(* IEC 61131-3 sources: SRCI/RobotLibrary/Library/Functions/Convert/TO_STRING, 78 files *)

(* ---- ABORTING_MODE_TO_STRING.st ---- *)
FUNCTION ABORTING_MODE_TO_STRING : STRING
// -------------------------------------------------------------------------
//  SRCI Robot Library
// -------------------------------------------------------------------------
//
//  Object:      ABORTING_MODE_TO_STRING
//  Author:      Thorsten Brach
//  Date:        2025-02-23
//
//  Description:
//
//
//  Copyright:
//    (C) 2025 Thorsten Brach. All rights reserved
//             Licensed under the LGPL-3.0 license.
//
//  Disclaimer:
//    This project is provided without any guarantee and can be used for
//    private and commercial purposes. Any use is at the user’s
//    own risk and responsibility.
//
// -------------------------------------------------------------------------
VAR_INPUT
  /// AbortingMode
  Value : AbortingMode;
END_VAR

  CASE Value
  OF
    AbortingMode.BUFFER : ABORTING_MODE_TO_STRING := StrReplace('BUFFER ({0})','{0}' , SINT_TO_STRING(Value));
    AbortingMode.ABORT  : ABORTING_MODE_TO_STRING := StrReplace('ABORT ({0})' ,'{0}' , SINT_TO_STRING(Value));
  ELSE
    ABORTING_MODE_TO_STRING := CONCAT('ABORTING_MODE_TO_STRING Function: Error -> no parsing for value ', SINT_TO_STRING(Value));
  END_CASE

END_FUNCTION

(* ---- ALARM_MESSAGE_TO_STRING.st ---- *)
FUNCTION ALARM_MESSAGE_TO_STRING : STRING(RobotLibraryParameter.MESSAGE_TEXT_LEN)
// -------------------------------------------------------------------------
//  SRCI Robot Library
// -------------------------------------------------------------------------
//
//  Object:      ALARM_MESSAGE_TO_STRING
//  Author:      Thorsten Brach
//  Date:        2025-03-31
//
//  Description:
//
//
//  Copyright:
//    (C) 2025 Thorsten Brach. All rights reserved
//             Licensed under the LGPL-3.0 license.
//
//  Disclaimer:
//    This project is provided without any guarantee and can be used for
//    private and commercial purposes. Any use is at the user’s
//    own risk and responsibility.
//
// -------------------------------------------------------------------------
VAR_INPUT
  /// AlarmMessag
  Message : AlarmMessage;
END_VAR
VAR CONSTANT
  /// Carrage return and line feed
  CRLF       : STRING := '$R$N';
END_VAR

  ALARM_MESSAGE_TO_STRING := CONCAT    (ALARM_MESSAGE_TO_STRING, DATE_TO_STRING(Message.Timestamp.SystemDate));
  ALARM_MESSAGE_TO_STRING := CONCAT    (ALARM_MESSAGE_TO_STRING, '-');
  ALARM_MESSAGE_TO_STRING := CONCAT    (ALARM_MESSAGE_TO_STRING, TOD_TO_STRING (Message.Timestamp.SystemTime));
  ALARM_MESSAGE_TO_STRING := StrReplace(ALARM_MESSAGE_TO_STRING, 'TOD#','' );
  ALARM_MESSAGE_TO_STRING := StrReplace(ALARM_MESSAGE_TO_STRING, 'D#', '' );
  ALARM_MESSAGE_TO_STRING := CONCAT    (ALARM_MESSAGE_TO_STRING, ':');
  ALARM_MESSAGE_TO_STRING := CONCAT    (ALARM_MESSAGE_TO_STRING, MESSAGE_TYPE_TO_STRING(Value := Message.MessageType, AlignString := TRUE));
  ALARM_MESSAGE_TO_STRING := CONCAT    (ALARM_MESSAGE_TO_STRING, ':');
  ALARM_MESSAGE_TO_STRING := CONCAT    (ALARM_MESSAGE_TO_STRING, SEVERITY_TO_STRING    ( Value := Message.Severity  , AlignString := TRUE));
  ALARM_MESSAGE_TO_STRING := CONCAT    (ALARM_MESSAGE_TO_STRING, ':');
  ALARM_MESSAGE_TO_STRING := CONCAT    (ALARM_MESSAGE_TO_STRING, DWORD_TO_STRING(Message.MessageCode));
  ALARM_MESSAGE_TO_STRING := CONCAT    (ALARM_MESSAGE_TO_STRING, ':');
  ALARM_MESSAGE_TO_STRING := CONCAT    (ALARM_MESSAGE_TO_STRING, Message.MessageText);
  ALARM_MESSAGE_TO_STRING := CONCAT    (ALARM_MESSAGE_TO_STRING, CRLF);

END_FUNCTION

(* ---- AREA_TYPE_TO_STRING.st ---- *)
FUNCTION AREA_TYPE_TO_STRING : STRING
// -------------------------------------------------------------------------
//  SRCI Robot Library
// -------------------------------------------------------------------------
//
//  Object:      AREA_TYPE_TO_STRING
//  Author:      Thorsten Brach
//  Date:        2025-02-01
//
//  Description:
//
//
//  Copyright:
//    (C) 2025 Thorsten Brach. All rights reserved
//             Licensed under the LGPL-3.0 license.
//
//  Disclaimer:
//    This project is provided without any guarantee and can be used for
//    private and commercial purposes. Any use is at the user’s
//    own risk and responsibility.
//
// -------------------------------------------------------------------------
VAR_INPUT
  /// AreaType
  Value : AreaType;
END_VAR

  CASE Value
  OF
    AreaType.AXES     : AREA_TYPE_TO_STRING := StrReplace('AXES ({0})'     ,'{0}' , USINT_TO_STRING(Value));
    AreaType.BOX      : AREA_TYPE_TO_STRING := StrReplace('BOX ({0})'      ,'{0}' , USINT_TO_STRING(Value));
    AreaType.CYLINDER : AREA_TYPE_TO_STRING := StrReplace('CYLINDER ({0})' ,'{0}' , USINT_TO_STRING(Value));
    AreaType.SPHERE   : AREA_TYPE_TO_STRING := StrReplace('SPHERE ({0})'   ,'{0}' , USINT_TO_STRING(Value));
  ELSE
    AREA_TYPE_TO_STRING := CONCAT('AREA_TYPE_TO_STRING Function: Error -> no parsing for value ', USINT_TO_STRING(Value));
  END_CASE

END_FUNCTION

(* ---- ARM_CONFIG_ELBOW_TO_STRING.st ---- *)
FUNCTION ARM_CONFIG_ELBOW_TO_STRING : STRING
// -------------------------------------------------------------------------
//  SRCI Robot Library
// -------------------------------------------------------------------------
//
//  Object:      ARM_CONFIG_ELBOW_TO_STRING
//  Author:      Thorsten Brach
//  Date:        2025-02-04
//
//  Description:
//
//
//  Copyright:
//    (C) 2025 Thorsten Brach. All rights reserved
//             Licensed under the LGPL-3.0 license.
//
//  Disclaimer:
//    This project is provided without any guarantee and can be used for
//    private and commercial purposes. Any use is at the user’s
//    own risk and responsibility.
//
// -------------------------------------------------------------------------
VAR_INPUT
  /// ArmConfigElbow
  Value : ArmConfigElbow;
END_VAR

  CASE Value
  OF
    ArmConfigElbow.USE_CONFIG : ARM_CONFIG_ELBOW_TO_STRING := StrReplace('Elbow = USE_CONFIG ({0})','{0}' , INT_TO_STRING(Value));
    ArmConfigElbow.SAME       : ARM_CONFIG_ELBOW_TO_STRING := StrReplace('Elbow = SAME ({0})'      ,'{0}' , INT_TO_STRING(Value));
    ArmConfigElbow.FREE       : ARM_CONFIG_ELBOW_TO_STRING := StrReplace('Elbow = FREE ({0})'      ,'{0}' , INT_TO_STRING(Value));
    ArmConfigElbow.DOWN       : ARM_CONFIG_ELBOW_TO_STRING := StrReplace('Elbow = DOWN ({0})'      ,'{0}' , INT_TO_STRING(Value));
    ArmConfigElbow.UP         : ARM_CONFIG_ELBOW_TO_STRING := StrReplace('Elbow = UP ({0})'        ,'{0}' , INT_TO_STRING(Value));
  ELSE
    ARM_CONFIG_ELBOW_TO_STRING := CONCAT('ARM_CONFIG_ELBOW_TO_STRING Function: Error -> no parsing for value ', INT_TO_STRING(Value));
  END_CASE

END_FUNCTION

(* ---- ARM_CONFIG_SHOULDER_TO_STRING.st ---- *)
FUNCTION ARM_CONFIG_SHOULDER_TO_STRING : STRING
// -------------------------------------------------------------------------
//  SRCI Robot Library
// -------------------------------------------------------------------------
//
//  Object:      ARM_CONFIG_SHOULDER_TO_STRING
//  Author:      Thorsten Brach
//  Date:        2025-02-04
//
//  Description:
//
//
//  Copyright:
//    (C) 2025 Thorsten Brach. All rights reserved
//             Licensed under the LGPL-3.0 license.
//
//  Disclaimer:
//    This project is provided without any guarantee and can be used for
//    private and commercial purposes. Any use is at the user’s
//    own risk and responsibility.
//
// -------------------------------------------------------------------------
VAR_INPUT
  /// ArmConfigShoulder
  Value : ArmConfigShoulder;
END_VAR

  CASE Value
  OF
    ArmConfigShoulder.USE_CONFIG : ARM_CONFIG_SHOULDER_TO_STRING := StrReplace('Shoulder = USE_CONFIG ({0})','{0}' , INT_TO_STRING(Value));
    ArmConfigShoulder.SAME       : ARM_CONFIG_SHOULDER_TO_STRING := StrReplace('Shoulder = SAME ({0})'      ,'{0}' , INT_TO_STRING(Value));
    ArmConfigShoulder.FREE       : ARM_CONFIG_SHOULDER_TO_STRING := StrReplace('Shoulder = FREE ({0})'      ,'{0}' , INT_TO_STRING(Value));
    ArmConfigShoulder.BACK       : ARM_CONFIG_SHOULDER_TO_STRING := StrReplace('Shoulder = BACK ({0})'      ,'{0}' , INT_TO_STRING(Value));
    ArmConfigShoulder.FRONT      : ARM_CONFIG_SHOULDER_TO_STRING := StrReplace('Shoulder = FRONT ({0})'     ,'{0}' , INT_TO_STRING(Value));
  ELSE
    ARM_CONFIG_SHOULDER_TO_STRING := CONCAT('ARM_CONFIG_SHOULDER_TO_STRING Function: Error -> no parsing for value ', INT_TO_STRING(Value));
  END_CASE

END_FUNCTION

(* ---- ARM_CONFIG_TO_STRING.st ---- *)
FUNCTION ARM_CONFIG_TO_STRING : STRING
// -------------------------------------------------------------------------
//  SRCI Robot Library
// -------------------------------------------------------------------------
//
//  Object:      ARM_CONFIG_TO_STRING
//  Author:      Thorsten Brach
//  Date:        2025-01-23
//
//  Description:
//
//
//  Copyright:
//    (C) 2025 Thorsten Brach. All rights reserved
//             Licensed under the LGPL-3.0 license.
//
//  Disclaimer:
//    This project is provided without any guarantee and can be used for
//    private and commercial purposes. Any use is at the user’s
//    own risk and responsibility.
//
// -------------------------------------------------------------------------
VAR_INPUT
  /// ArmConfigParameter
  Value : ArmConfigParameter;
END_VAR

VAR
  /// temporary byte
 _tmpByte : BYTE;
END_VAR

  Value := Value;

  _tmpByte.0 := Value.Shoulder = ArmConfigShoulder.USE_CONFIG;
  _tmpByte.1 := Value.Elbow    = ArmConfigElbow   .USE_CONFIG;
  _tmpByte.2 := Value.Wrist    = ArmConfigWrist   .USE_CONFIG;

  ARM_CONFIG_TO_STRING := BYTE_TO_STRING_BIN(_tmpByte);

END_FUNCTION

(* ---- ARM_CONFIG_WRIST_TO_STRING.st ---- *)
FUNCTION ARM_CONFIG_WRIST_TO_STRING : STRING
// -------------------------------------------------------------------------
//  SRCI Robot Library
// -------------------------------------------------------------------------
//
//  Object:      ARM_CONFIG_WRIST_TO_STRING
//  Author:      Thorsten Brach
//  Date:        2025-02-04
//
//  Description:
//
//
//  Copyright:
//    (C) 2025 Thorsten Brach. All rights reserved
//             Licensed under the LGPL-3.0 license.
//
//  Disclaimer:
//    This project is provided without any guarantee and can be used for
//    private and commercial purposes. Any use is at the user’s
//    own risk and responsibility.
//
// -------------------------------------------------------------------------
VAR_INPUT
  /// ArmConfigWrist
  Value : ArmConfigWrist;
END_VAR

  CASE Value
  OF
    ArmConfigWrist.USE_CONFIG : ARM_CONFIG_WRIST_TO_STRING := StrReplace('Wrist = USE_CONFIG ({0})','{0}' , INT_TO_STRING(Value));
    ArmConfigWrist.SAME       : ARM_CONFIG_WRIST_TO_STRING := StrReplace('Wrist = SAME ({0})'      ,'{0}' , INT_TO_STRING(Value));
    ArmConfigWrist.FREE       : ARM_CONFIG_WRIST_TO_STRING := StrReplace('Wrist = FREE ({0})'      ,'{0}' , INT_TO_STRING(Value));
    ArmConfigWrist.FLIP       : ARM_CONFIG_WRIST_TO_STRING := StrReplace('Wrist = FLIP ({0})'      ,'{0}' , INT_TO_STRING(Value));
    ArmConfigWrist.NON_FLIP   : ARM_CONFIG_WRIST_TO_STRING := StrReplace('Wrist = NON_FLIP ({0})'  ,'{0}' , INT_TO_STRING(Value));
  ELSE
    ARM_CONFIG_WRIST_TO_STRING := CONCAT('ARM_CONFIG_WRIST_TO_STRING Function: Error -> no parsing for value ', INT_TO_STRING(Value));
  END_CASE

END_FUNCTION

(* ---- BLENDING_MODE_TO_STRING.st ---- *)
FUNCTION BLENDING_MODE_TO_STRING : STRING
// -------------------------------------------------------------------------
//  SRCI Robot Library
// -------------------------------------------------------------------------
//
//  Object:      BLENDING_MODE_TO_STRING
//  Author:      Thorsten Brach
//  Date:        2025-01-23
//
//  Description:
//
//
//  Copyright:
//    (C) 2025 Thorsten Brach. All rights reserved
//             Licensed under the LGPL-3.0 license.
//
//  Disclaimer:
//    This project is provided without any guarantee and can be used for
//    private and commercial purposes. Any use is at the user’s
//    own risk and responsibility.
//
// -------------------------------------------------------------------------
VAR_INPUT
  /// BlendingMode
  Value : BlendingMode;
END_VAR

  CASE Value
  OF
    BlendingMode.EXACT_STOP           : BLENDING_MODE_TO_STRING := StrReplace('EXACT_STOP ({0})','{0}'           , USINT_TO_STRING(Value));
    BlendingMode.DEFINED_VELOCITY     : BLENDING_MODE_TO_STRING := StrReplace('DEFINED_VELOCITY ({0})','{0}'     , USINT_TO_STRING(Value));
    BlendingMode.CORNER_DISTANCE      : BLENDING_MODE_TO_STRING := StrReplace('CORNER_DISTANCE ({0})','{0}'      , USINT_TO_STRING(Value));
    BlendingMode.MAX_CORNER_DEVIATION : BLENDING_MODE_TO_STRING := StrReplace('MAX_CORNER_DEVIATION ({0})','{0}' , USINT_TO_STRING(Value));
    BlendingMode.CORNER_DISTANCE_2R   : BLENDING_MODE_TO_STRING := StrReplace('CORNER_DISTANCE_2R ({0})','{0}'   , USINT_TO_STRING(Value));
    BlendingMode.RAMP_OVERLAP         : BLENDING_MODE_TO_STRING := StrReplace('RAMP_OVERLAP ({0})','{0}'         , USINT_TO_STRING(Value));
    BlendingMode.CORNER_DISTANCE_1R   : BLENDING_MODE_TO_STRING := StrReplace('CORNER_DISTANCE_1R ({0})','{0}'   , USINT_TO_STRING(Value));
  ELSE
    BLENDING_MODE_TO_STRING := CONCAT('BLENDING_MODE_TO_STRING Function: Error -> no parsing for value ', USINT_TO_STRING(Value));
  END_CASE

END_FUNCTION

(* ---- BYTE_TO_STRING_BIN.st ---- *)
FUNCTION BYTE_TO_STRING_BIN : STRING
// -------------------------------------------------------------------------
//  SRCI Robot Library
// -------------------------------------------------------------------------
//
//  Object:      BYTE_TO_STRING_BIN
//  Author:      Thorsten Brach
//  Date:        2025-01-20
//
//  Description:
//    Converts a BYTE to a STRING with binary notation
//
//  Copyright:
//    (C) 2024 Thorsten Brach. All rights reserved
//             Licensed under the LGPL-3.0 license.
//
//  Disclaimer:
//    This project is provided without any guarantee and can be used for
//    private and commercial purposes. Any use is at the user’s
//    own risk and responsibility.
//
// -------------------------------------------------------------------------
VAR_INPUT
 /// Value to convert
 Value : BYTE;
END_VAR

  BYTE_TO_STRING_BIN := '2#';

  IF (Value.7)
  THEN
    BYTE_TO_STRING_BIN := CONCAT(BYTE_TO_STRING_BIN, '1');
  ELSE
    BYTE_TO_STRING_BIN := CONCAT(BYTE_TO_STRING_BIN, '0');
  END_IF

  IF (Value.6)
  THEN
    BYTE_TO_STRING_BIN := CONCAT(BYTE_TO_STRING_BIN, '1');
  ELSE
    BYTE_TO_STRING_BIN := CONCAT(BYTE_TO_STRING_BIN, '0');
  END_IF

  IF (Value.5)
  THEN
    BYTE_TO_STRING_BIN := CONCAT(BYTE_TO_STRING_BIN, '1');
  ELSE
    BYTE_TO_STRING_BIN := CONCAT(BYTE_TO_STRING_BIN, '0');
  END_IF

  IF (Value.4)
  THEN
    BYTE_TO_STRING_BIN := CONCAT(BYTE_TO_STRING_BIN, '1_');
  ELSE
    BYTE_TO_STRING_BIN := CONCAT(BYTE_TO_STRING_BIN, '0_');
  END_IF

  IF (Value.3)
  THEN
    BYTE_TO_STRING_BIN := CONCAT(BYTE_TO_STRING_BIN, '1');
  ELSE
    BYTE_TO_STRING_BIN := CONCAT(BYTE_TO_STRING_BIN, '0');
  END_IF

  IF (Value.2)
  THEN
    BYTE_TO_STRING_BIN := CONCAT(BYTE_TO_STRING_BIN, '1');
  ELSE
    BYTE_TO_STRING_BIN := CONCAT(BYTE_TO_STRING_BIN, '0');
  END_IF

  IF (Value.1)
  THEN
    BYTE_TO_STRING_BIN := CONCAT(BYTE_TO_STRING_BIN, '1');
  ELSE
    BYTE_TO_STRING_BIN := CONCAT(BYTE_TO_STRING_BIN, '0');
  END_IF

  IF (Value.0)
  THEN
    BYTE_TO_STRING_BIN := CONCAT(BYTE_TO_STRING_BIN, '1');
  ELSE
    BYTE_TO_STRING_BIN := CONCAT(BYTE_TO_STRING_BIN, '0');
  END_IF

  BYTE_TO_STRING_BIN := CONCAT(BYTE_TO_STRING_BIN, ' (');
  BYTE_TO_STRING_BIN := CONCAT(BYTE_TO_STRING_BIN, WORD_TO_STRING(Value));
  BYTE_TO_STRING_BIN := CONCAT(BYTE_TO_STRING_BIN, ')');

END_FUNCTION

(* ---- CIRC_MODE_TO_STRING.st ---- *)
FUNCTION CIRC_MODE_TO_STRING : STRING
// -------------------------------------------------------------------------
//  SRCI Robot Library
// -------------------------------------------------------------------------
//
//  Object:      CIRC_MODE_TO_STRING
//  Author:      Thorsten Brach
//  Date:        2025-01-30
//
//  Description:
//
//
//  Copyright:
//    (C) 2025 Thorsten Brach. All rights reserved
//             Licensed under the LGPL-3.0 license.
//
//  Disclaimer:
//    This project is provided without any guarantee and can be used for
//    private and commercial purposes. Any use is at the user’s
//    own risk and responsibility.
//
// -------------------------------------------------------------------------
VAR_INPUT
  /// CircMode
  Value : CircMode;
END_VAR

  CASE Value
  OF
    CircMode.BORDER            : CIRC_MODE_TO_STRING := StrReplace('BORDER ({0})'            ,'{0}' , SINT_TO_STRING(Value));
    CircMode.CENTER            : CIRC_MODE_TO_STRING := StrReplace('CENTER ({0})'            ,'{0}' , SINT_TO_STRING(Value));
    CircMode.CENTER_WITH_ANGLE : CIRC_MODE_TO_STRING := StrReplace('CENTER_WITH_ANGLE ({0})' ,'{0}' , SINT_TO_STRING(Value));
    CircMode.RADIUS            : CIRC_MODE_TO_STRING := StrReplace('RADIUS ({0})'            ,'{0}' , SINT_TO_STRING(Value));
  ELSE
    CIRC_MODE_TO_STRING := CONCAT('CIRC_MODE_TO_STRING Function: Error -> no parsing for value ', SINT_TO_STRING(Value));
  END_CASE

END_FUNCTION

(* ---- CIRC_PLANE_TO_STRING.st ---- *)
FUNCTION CIRC_PLANE_TO_STRING : STRING
// -------------------------------------------------------------------------
//  SRCI Robot Library
// -------------------------------------------------------------------------
//
//  Object:      CIRC_PLANE_TO_STRING
//  Author:      Thorsten Brach
//  Date:        2025-01-30
//
//  Description:
//
//
//  Copyright:
//    (C) 2025 Thorsten Brach. All rights reserved
//             Licensed under the LGPL-3.0 license.
//
//  Disclaimer:
//    This project is provided without any guarantee and can be used for
//    private and commercial purposes. Any use is at the user’s
//    own risk and responsibility.
//
// -------------------------------------------------------------------------
VAR_INPUT
  /// CircPlane
  Value : CircPlane;
END_VAR

  CASE Value
  OF
    CircPlane.XZ_PLANE : CIRC_PLANE_TO_STRING := StrReplace('XZ_PLANE ({0})' ,'{0}' , SINT_TO_STRING(Value));
    CircPlane.YZ_PLANE : CIRC_PLANE_TO_STRING := StrReplace('YZ_PLANE ({0})' ,'{0}' , SINT_TO_STRING(Value));
    CircPlane.XY_PLANE : CIRC_PLANE_TO_STRING := StrReplace('XY_PLANE ({0})' ,'{0}' , SINT_TO_STRING(Value));
  ELSE
    CIRC_PLANE_TO_STRING := CONCAT('CIRC_PLANE_TO_STRING Function: Error -> no parsing for value ', SINT_TO_STRING(Value));
  END_CASE

END_FUNCTION

(* ---- CMD_MESSAGE_STATE_TO_STRING.st ---- *)
FUNCTION CMD_MESSAGE_STATE_TO_STRING : STRING
// -------------------------------------------------------------------------
//  SRCI Robot Library
// -------------------------------------------------------------------------
//
//  Object:      CMD_MESSAGE_STATE_TO_STRING
//  Author:      Thorsten Brach
//  Date:        2024-11-16
//
//  Description:
//
//
//  Copyright:
//    (C) 2024 Thorsten Brach. All rights reserved
//             Licensed under the LGPL-3.0 license.
//
//  Disclaimer:
//    This project is provided without any guarantee and can be used for
//    private and commercial purposes. Any use is at the user’s
//    own risk and responsibility.
//
// -------------------------------------------------------------------------
VAR_INPUT
  /// Command message state
  Value : CmdMessageState;
END_VAR

  CASE Value
  OF
    CmdMessageState.EMPTY               : CMD_MESSAGE_STATE_TO_STRING := StrReplace('EMPTY ({0})'              ,'{0}', USINT_TO_STRING(Value));
    CmdMessageState.CREATED             : CMD_MESSAGE_STATE_TO_STRING := StrReplace('CREATED ({0})'            ,'{0}', USINT_TO_STRING(Value));
    CmdMessageState.BUFFERED            : CMD_MESSAGE_STATE_TO_STRING := StrReplace('BUFFERED ({0})'           ,'{0}', USINT_TO_STRING(Value));
    CmdMessageState.BUFFERED_IN_PLANNER : CMD_MESSAGE_STATE_TO_STRING := StrReplace('BUFFERED_IN_PLANNER ({0})','{0}', USINT_TO_STRING(Value));
    CmdMessageState.ACTIVE              : CMD_MESSAGE_STATE_TO_STRING := StrReplace('ACTIVE ({0})'             ,'{0}', USINT_TO_STRING(Value));
    CmdMessageState.INTERRUPTED         : CMD_MESSAGE_STATE_TO_STRING := StrReplace('INTERRUPTED ({0})'        ,'{0}', USINT_TO_STRING(Value));
    CmdMessageState.ABORT_REQUEST       : CMD_MESSAGE_STATE_TO_STRING := StrReplace('ABORT_REQUEST ({0})'      ,'{0}', USINT_TO_STRING(Value));
    CmdMessageState.DONE                : CMD_MESSAGE_STATE_TO_STRING := StrReplace('DONE ({0})'               ,'{0}', USINT_TO_STRING(Value));
    CmdMessageState.ABORTED             : CMD_MESSAGE_STATE_TO_STRING := StrReplace('ABORTED ({0})'            ,'{0}', USINT_TO_STRING(Value));
    CmdMessageState.ERROR               : CMD_MESSAGE_STATE_TO_STRING := StrReplace('ERROR ({0})'              ,'{0}', USINT_TO_STRING(Value));
  ELSE
    CMD_MESSAGE_STATE_TO_STRING := CONCAT('CMD_MESSAGE_STATE_TO_STRING Function: Error -> no parsing for value ', USINT_TO_STRING(Value));
  END_CASE

END_FUNCTION

(* ---- CMD_TYPE_TO_STRING.st ---- *)
FUNCTION CMD_TYPE_TO_STRING : String
// -------------------------------------------------------------------------
//  SRCI Robot Library
// -------------------------------------------------------------------------
//
//  Object:      CMD_TYPE_TO_STRING
//  Author:      Thorsten Brach
//  Date:        2024-11-16
//
//  Description:
//
//
//  Copyright:
//    (C) 2024 Thorsten Brach. All rights reserved
//             Licensed under the LGPL-3.0 license.
//
//  Disclaimer:
//    This project is provided without any guarantee and can be used for
//    private and commercial purposes. Any use is at the user’s
//    own risk and responsibility.
//
// -------------------------------------------------------------------------
VAR_INPUT
  /// command type
  Value : CmdType;
END_VAR

  CASE Value
  OF
    CmdType.RobotTask                   : CMD_TYPE_TO_STRING := StrReplace('RobotTask ({0})','{0}'                  , UINT_TO_STRING(CmdType.RobotTask));

    CmdType.ReadRobotData               : CMD_TYPE_TO_STRING := StrReplace('ReadRobotData ({0})','{0}'              , UINT_TO_STRING(CmdType.ReadRobotData));

    CmdType.EnableRobot                 : CMD_TYPE_TO_STRING := StrReplace('EnableRobot ({0})','{0}'                , UINT_TO_STRING(CmdType.EnableRobot));

    CmdType.GroupReset                  : CMD_TYPE_TO_STRING := StrReplace('GroupReset ({0})','{0}'                 , UINT_TO_STRING(CmdType.GroupReset));

    CmdType.ReadActualPosition          : CMD_TYPE_TO_STRING := StrReplace('ReadActualPosition ({0})','{0}'         , UINT_TO_STRING(CmdType.ReadActualPosition));

    CmdType.ReadActualPositionCyclic    : CMD_TYPE_TO_STRING := StrReplace('ReadActualPositionCyclic ({0})','{0}'   , UINT_TO_STRING(CmdType.ReadActualPositionCyclic));

    CmdType.ReadDHParameter             : CMD_TYPE_TO_STRING := StrReplace('ReadDHParameter ({0})','{0}'            , UINT_TO_STRING(CmdType.ReadDHParameter));

    CmdType.RestartController           : CMD_TYPE_TO_STRING := StrReplace('RestartController ({0})','{0}'          , UINT_TO_STRING(CmdType.RestartController));

    CmdType.ReadActualTCPVelocity       : CMD_TYPE_TO_STRING := StrReplace('ReadActualTCPVelocity ({0})','{0}'      , UINT_TO_STRING(CmdType.ReadActualTCPVelocity));

    CmdType.UserLogin                   : CMD_TYPE_TO_STRING := StrReplace('UserLogin ({0})','{0}'                  , UINT_TO_STRING(CmdType.UserLogin));

    CmdType.SwitchLanguage              : CMD_TYPE_TO_STRING := StrReplace('SwitchLanguage ({0})','{0}'             , UINT_TO_STRING(CmdType.SwitchLanguage));

    CmdType.ExchangeConfiguration       : CMD_TYPE_TO_STRING := StrReplace('ExchangeConfiguration ({0})','{0}'      , UINT_TO_STRING(CmdType.ExchangeConfiguration));

    CmdType.SetSequence                 : CMD_TYPE_TO_STRING := StrReplace('SetSequence ({0})','{0}'                , UINT_TO_STRING(CmdType.SetSequence));

    CmdType.ChangeSpeedOverride         : CMD_TYPE_TO_STRING := StrReplace('ChangeSpeedOverride ({0})','{0}'        , UINT_TO_STRING(CmdType.ChangeSpeedOverride));

    CmdType.ReadMessages                : CMD_TYPE_TO_STRING := StrReplace('ReadMessages ({0})','{0}'               , UINT_TO_STRING(CmdType.ReadMessages));

    CmdType.ReadRobotReferenceDynamics  : CMD_TYPE_TO_STRING := StrReplace('ReadRobotReferenceDynamics ({0})','{0}' , UINT_TO_STRING(CmdType.ReadRobotReferenceDynamics));

    CmdType.WriteFrameData              : CMD_TYPE_TO_STRING := StrReplace('WriteFrameData ({0})','{0}'             , UINT_TO_STRING(CmdType.WriteFrameData));

    CmdType.WriteToolData               : CMD_TYPE_TO_STRING := StrReplace('WriteToolData ({0})','{0}'              , UINT_TO_STRING(CmdType.WriteToolData));

    CmdType.WriteLoadData               : CMD_TYPE_TO_STRING := StrReplace('WriteLoadData ({0})','{0}'              , UINT_TO_STRING(CmdType.WriteLoadData));

    CmdType.WriteRobotReferenceDynamics : CMD_TYPE_TO_STRING := StrReplace('WriteRobotReferenceDynamics ({0})','{0}', UINT_TO_STRING(CmdType.WriteRobotReferenceDynamics));

    CmdType.WriteRobotDefaultDynamics   : CMD_TYPE_TO_STRING := StrReplace('WriteRobotDefaultDynamics ({0})'  ,'{0}', UINT_TO_STRING(CmdType.WriteRobotDefaultDynamics));

    CmdType.ReadRobotDefaultDynamics    : CMD_TYPE_TO_STRING := StrReplace('ReadRobotDefaultDynamics ({0})'   ,'{0}', UINT_TO_STRING(CmdType.ReadRobotDefaultDynamics));

    CmdType.ReadFrameData               : CMD_TYPE_TO_STRING := StrReplace('ReadFrameData ({0})'              ,'{0}', UINT_TO_STRING(CmdType.ReadFrameData));

    CmdType.ReadToolData                : CMD_TYPE_TO_STRING := StrReplace('ReadToolData ({0})','{0}'               , UINT_TO_STRING(CmdType.ReadToolData));

    CmdType.ReadLoadData                : CMD_TYPE_TO_STRING := StrReplace('ReadLoadData ({0})','{0}'               , UINT_TO_STRING(CmdType.ReadLoadData));

    CmdType.ReadRobotSWLimits           : CMD_TYPE_TO_STRING := StrReplace('ReadRobotSWLimits ({0})','{0}'          , UINT_TO_STRING(CmdType.ReadRobotSWLimits));

    CmdType.WriteRobotSWLimits          : CMD_TYPE_TO_STRING := StrReplace('WriteRobotSWLimits ({0})','{0}'         , UINT_TO_STRING(CmdType.WriteRobotSWLimits));

    CmdType.SetOperationMode            : CMD_TYPE_TO_STRING := StrReplace('SetOperationMode ({0})','{0}'           , UINT_TO_STRING(CmdType.SetOperationMode));

    CmdType.ReadWorkArea                : CMD_TYPE_TO_STRING := StrReplace('ReadWorkArea ({0})','{0}'               , UINT_TO_STRING(CmdType.ReadWorkArea));

    CmdType.WriteWorkArea               : CMD_TYPE_TO_STRING := StrReplace('WriteWorkArea ({0})','{0}'              , UINT_TO_STRING(CmdType.WriteWorkArea));

    CmdType.ActivateWorkArea            : CMD_TYPE_TO_STRING := StrReplace('ActivateWorkArea ({0})','{0}'           , UINT_TO_STRING(CmdType.ActivateWorkArea));

    CmdType.MonitorWorkArea             : CMD_TYPE_TO_STRING := StrReplace('MonitorWorkArea ({0})','{0}'            , UINT_TO_STRING(CmdType.MonitorWorkArea));

    CmdType.GroupJog                    : CMD_TYPE_TO_STRING := StrReplace('GroupJog ({0})','{0}'                   , UINT_TO_STRING(CmdType.GroupJog));

    CmdType.MoveLinearAbsolute          : CMD_TYPE_TO_STRING := StrReplace('MoveLinearAbsolute ({0})','{0}'         , UINT_TO_STRING(CmdType.MoveLinearAbsolute));

    CmdType.MoveDirectAbsolute          : CMD_TYPE_TO_STRING := StrReplace('MoveDirectAbsolute ({0})','{0}'         , UINT_TO_STRING(CmdType.MoveDirectAbsolute));

    CmdType.MoveAxesAbsolute            : CMD_TYPE_TO_STRING := StrReplace('MoveAxesAbsolute ({0})','{0}'           , UINT_TO_STRING(CmdType.MoveAxesAbsolute));

    CmdType.GroupStop                   : CMD_TYPE_TO_STRING := StrReplace('GroupStop ({0})','{0}'                  , UINT_TO_STRING(CmdType.GroupStop));

    CmdType.GroupInterrupt              : CMD_TYPE_TO_STRING := StrReplace('GroupInterrupt ({0})','{0}'             , UINT_TO_STRING(CmdType.GroupInterrupt));

    CmdType.GroupContinue               : CMD_TYPE_TO_STRING := StrReplace('GroupContinue ({0})','{0}'              , UINT_TO_STRING(CmdType.GroupContinue));

    CmdType.MoveLinearRelative          : CMD_TYPE_TO_STRING := StrReplace('MoveLinearRelative ({0})','{0}'         , UINT_TO_STRING(CmdType.MoveLinearRelative));

    CmdType.MoveDirectRelative          : CMD_TYPE_TO_STRING := StrReplace('MoveDirectRelative ({0})','{0}'         , UINT_TO_STRING(CmdType.MoveDirectRelative));

    CmdType.MoveAxesRelative            : CMD_TYPE_TO_STRING := StrReplace('MoveAxesRelative ({0})','{0}'           , UINT_TO_STRING(CmdType.MoveAxesRelative));

    CmdType.ReturnToPrimary             : CMD_TYPE_TO_STRING := StrReplace('ReturnToPrimary ({0})','{0}'            , UINT_TO_STRING(CmdType.ReturnToPrimary));

    CmdType.MoveCircularAbsolute        : CMD_TYPE_TO_STRING := StrReplace('MoveCircularAbsolute ({0})','{0}'       , UINT_TO_STRING(CmdType.MoveCircularAbsolute));

    CmdType.MoveCircularRelative        : CMD_TYPE_TO_STRING := StrReplace('MoveCircularRelative ({0})','{0}'       , UINT_TO_STRING(CmdType.MoveCircularRelative));

    CmdType.MoveLinearOffset            : CMD_TYPE_TO_STRING := StrReplace('MoveLinearOffset ({0})','{0}'           , UINT_TO_STRING(CmdType.MoveLinearOffset));

    CmdType.MoveDirectOffset            : CMD_TYPE_TO_STRING := StrReplace('MoveDirectOffset ({0})','{0}'           , UINT_TO_STRING(CmdType.MoveDirectOffset));

    CmdType.WaitTime                    : CMD_TYPE_TO_STRING := StrReplace('WaitTime ({0})','{0}'                   , UINT_TO_STRING(CmdType.WaitTime));

    CmdType.MoveApproachLinear          : CMD_TYPE_TO_STRING := StrReplace('MoveApproachLinear ({0})','{0}'         , UINT_TO_STRING(CmdType.MoveApproachLinear));

    CmdType.MoveDepartLinear            : CMD_TYPE_TO_STRING := StrReplace('MoveDepartLinear ({0})','{0}'           , UINT_TO_STRING(CmdType.MoveDepartLinear));

    CmdType.MoveApproachDirect          : CMD_TYPE_TO_STRING := StrReplace('MoveApproachDirect ({0})','{0}'         , UINT_TO_STRING(CmdType.MoveApproachDirect));

    CmdType.MoveDepartDirect            : CMD_TYPE_TO_STRING := StrReplace('MoveDepartDirect ({0})','{0}'           , UINT_TO_STRING(CmdType.MoveDepartDirect));

    CmdType.SearchHardstop              : CMD_TYPE_TO_STRING := StrReplace('SearchHardstop ({0})','{0}'             , UINT_TO_STRING(CmdType.SearchHardstop));

    CmdType.SearchHardstopJ             : CMD_TYPE_TO_STRING := StrReplace('SearchHardstopJ ({0})','{0}'            , UINT_TO_STRING(CmdType.SearchHardstopJ));

    CmdType.MovePickPlaceLinear         : CMD_TYPE_TO_STRING := StrReplace('MovePickPlaceLinear ({0})','{0}'        , UINT_TO_STRING(CmdType.MovePickPlaceLinear));

    CmdType.MovePickPlaceDirect         : CMD_TYPE_TO_STRING := StrReplace('MovePickPlaceDirect ({0})','{0}'        , UINT_TO_STRING(CmdType.MovePickPlaceDirect));

    CmdType.ActivateConveyorTracking    : CMD_TYPE_TO_STRING := StrReplace('ActivateConveyorTracking ({0})','{0}'   , UINT_TO_STRING(CmdType.ActivateConveyorTracking));

    CmdType.RedefineTrackingPos         : CMD_TYPE_TO_STRING := StrReplace('RedefineTrackingPos ({0})','{0}'        , UINT_TO_STRING(CmdType.RedefineTrackingPos));

    CmdType.SyncToConveyor              : CMD_TYPE_TO_STRING := StrReplace('SyncToConveyor ({0})','{0}'             , UINT_TO_STRING(CmdType.SyncToConveyor));

    CmdType.ConfigureConveyor           : CMD_TYPE_TO_STRING := StrReplace('ConfigureConveyor ({0})','{0}'          , UINT_TO_STRING(CmdType.ConfigureConveyor));

    CmdType.MoveSuperImposed            : CMD_TYPE_TO_STRING := StrReplace('MoveSuperImposed ({0})','{0}'           , UINT_TO_STRING(CmdType.MoveSuperImposed));

    CmdType.MoveSuperImposedDynamic     : CMD_TYPE_TO_STRING := StrReplace('MoveSuperImposedDynamic ({0})','{0}'    , UINT_TO_STRING(CmdType.MoveSuperImposedDynamic));

    CmdType.ReadDigitalInputs           : CMD_TYPE_TO_STRING := StrReplace('ReadDigitalInputs ({0})','{0}'          , UINT_TO_STRING(CmdType.ReadDigitalInputs));

    CmdType.ReadDigitalOutputs          : CMD_TYPE_TO_STRING := StrReplace('ReadDigitalOutputs ({0})','{0}'         , UINT_TO_STRING(CmdType.ReadDigitalOutputs));

    CmdType.WriteDigitalOutputs         : CMD_TYPE_TO_STRING := StrReplace('WriteDigitalOutputs ({0})','{0}'        , UINT_TO_STRING(CmdType.WriteDigitalOutputs));

    CmdType.ReadIntegers                : CMD_TYPE_TO_STRING := StrReplace('ReadIntegers ({0})','{0}'               , UINT_TO_STRING(CmdType.ReadIntegers));

    CmdType.ReadReals                   : CMD_TYPE_TO_STRING := StrReplace('ReadReals ({0})','{0}'                  , UINT_TO_STRING(CmdType.ReadReals));

    CmdType.WriteIntegers               : CMD_TYPE_TO_STRING := StrReplace('WriteIntegers ({0})','{0}'              , UINT_TO_STRING(CmdType.WriteIntegers));

    CmdType.WriteReals                  : CMD_TYPE_TO_STRING := StrReplace('WriteReals ({0})','{0}'                 , UINT_TO_STRING(CmdType.WriteReals));

    CmdType.MoveLinearCam               : CMD_TYPE_TO_STRING := StrReplace('MoveLinearCam ({0})','{0}'              , UINT_TO_STRING(CmdType.MoveLinearCam));

    CmdType.MoveDirectCam               : CMD_TYPE_TO_STRING := StrReplace('MoveDirectCam ({0})','{0}'              , UINT_TO_STRING(CmdType.MoveDirectCam));

    CmdType.MoveCircularCam             : CMD_TYPE_TO_STRING := StrReplace('MoveCircularCam ({0})','{0}'            , UINT_TO_STRING(CmdType.MoveCircularCam));

    CmdType.ReadAnalogInput             : CMD_TYPE_TO_STRING := StrReplace('ReadAnalogInput ({0})','{0}'            , UINT_TO_STRING(CmdType.ReadAnalogInput));

    CmdType.ReadAnalogOutput            : CMD_TYPE_TO_STRING := StrReplace('ReadAnalogOutput ({0})','{0}'           , UINT_TO_STRING(CmdType.ReadAnalogOutput));

    CmdType.WriteAnalogOutput           : CMD_TYPE_TO_STRING := StrReplace('WriteAnalogOutput ({0})','{0}'          , UINT_TO_STRING(CmdType.WriteAnalogOutput));

    CmdType.MeasuringInput              : CMD_TYPE_TO_STRING := StrReplace('MeasuringInput ({0})','{0}'             , UINT_TO_STRING(CmdType.MeasuringInput));

    CmdType.AbortMeasuringInput         : CMD_TYPE_TO_STRING := StrReplace('AbortMeasuringInput ({0})','{0}'        , UINT_TO_STRING(CmdType.AbortMeasuringInput));

    CmdType.SetTriggerRegister          : CMD_TYPE_TO_STRING := StrReplace('SetTriggerRegister ({0})','{0}'         , UINT_TO_STRING(CmdType.SetTriggerRegister));

    CmdType.SetTriggerLimit             : CMD_TYPE_TO_STRING := StrReplace('SetTriggerLimit ({0})','{0}'            , UINT_TO_STRING(CmdType.SetTriggerLimit));

    CmdType.SetTriggerUser              : CMD_TYPE_TO_STRING := StrReplace('SetTriggerUser ({0})','{0}'             , UINT_TO_STRING(CmdType.SetTriggerUser));

    CmdType.SetTriggerError             : CMD_TYPE_TO_STRING := StrReplace('SetTriggerError ({0})','{0}'            , UINT_TO_STRING(CmdType.SetTriggerError));

    CmdType.ReactAtTrigger              : CMD_TYPE_TO_STRING := StrReplace('ReactAtTrigger ({0})','{0}'             , UINT_TO_STRING(CmdType.ReactAtTrigger));

    CmdType.WaitForTrigger              : CMD_TYPE_TO_STRING := StrReplace('WaitForTrigger ({0})','{0}'             , UINT_TO_STRING(CmdType.WaitForTrigger));

    CmdType.ReadSystemVariable          : CMD_TYPE_TO_STRING := StrReplace('ReadSystemVariable ({0})','{0}'         , UINT_TO_STRING(CmdType.ReadSystemVariable));

    CmdType.WriteSystemVariable         : CMD_TYPE_TO_STRING := StrReplace('WriteSystemVariable ({0})','{0}'        , UINT_TO_STRING(CmdType.WriteSystemVariable));

    CmdType.CalculateForwardKinematic   : CMD_TYPE_TO_STRING := StrReplace('CalculateForwardKinematic ({0})','{0}'  , UINT_TO_STRING(CmdType.CalculateForwardKinematic));

    CmdType.CalculateInverseKinematic   : CMD_TYPE_TO_STRING := StrReplace('CalculateInverseKinematic ({0})','{0}'  , UINT_TO_STRING(CmdType.CalculateInverseKinematic));

    CmdType.CalculateCartesianPosition  : CMD_TYPE_TO_STRING := StrReplace('CalculateCartesianPosition ({0})','{0}' , UINT_TO_STRING(CmdType.CalculateCartesianPosition));

    CmdType.CalculateTool               : CMD_TYPE_TO_STRING := StrReplace('CalculateTool ({0})','{0}'              , UINT_TO_STRING(CmdType.CalculateTool));

    CmdType.CalculateFrame              : CMD_TYPE_TO_STRING := StrReplace('CalculateFrame ({0})','{0}'             , UINT_TO_STRING(CmdType.CalculateFrame));

    CmdType.ActivateNextCommand         : CMD_TYPE_TO_STRING := StrReplace('ActivateNextCommand ({0})','{0}'        , UINT_TO_STRING(CmdType.ActivateNextCommand));

    CmdType.ShiftPosition               : CMD_TYPE_TO_STRING := StrReplace('ShiftPosition ({0})','{0}'              , UINT_TO_STRING(CmdType.ShiftPosition));

    CmdType.SetTriggerMotion            : CMD_TYPE_TO_STRING := StrReplace('SetTriggerMotion ({0})','{0}'           , UINT_TO_STRING(CmdType.SetTriggerMotion));

    CmdType.OpenBrake                   : CMD_TYPE_TO_STRING := StrReplace('OpenBrake ({0})','{0}'                  , UINT_TO_STRING(CmdType.OpenBrake));

    CmdType.CallSubprogram              : CMD_TYPE_TO_STRING := StrReplace('CallSubprogram ({0})','{0}'             , UINT_TO_STRING(CmdType.CallSubprogram));

    CmdType.WriteCallSubprogramCyclic   : CMD_TYPE_TO_STRING := StrReplace('WriteCallSubprogramCyclic ({0})','{0}'  , UINT_TO_STRING(CmdType.WriteCallSubprogramCyclic));

    CmdType.ReadCallSubprogramCyclic    : CMD_TYPE_TO_STRING := StrReplace('ReadCallSubprogramCyclic ({0})','{0}'   , UINT_TO_STRING(CmdType.ReadCallSubprogramCyclic));

    CmdType.StopSubprogram              : CMD_TYPE_TO_STRING := StrReplace('StopSubprogram ({0})','{0}'             , UINT_TO_STRING(CmdType.StopSubprogram));

    CmdType.PathAccuracyMode            : CMD_TYPE_TO_STRING := StrReplace('PathAccuracyMode ({0})','{0}'           , UINT_TO_STRING(CmdType.PathAccuracyMode));

    CmdType.AvoidSingularity            : CMD_TYPE_TO_STRING := StrReplace('AvoidSingularity ({0})','{0}'           , UINT_TO_STRING(CmdType.AvoidSingularity));

    CmdType.ForceControl                : CMD_TYPE_TO_STRING := StrReplace('ForceControl ({0})','{0}'               , UINT_TO_STRING(CmdType.ForceControl));

    CmdType.ForceLimit                  : CMD_TYPE_TO_STRING := StrReplace('ForceLimit ({0})','{0}'                 , UINT_TO_STRING(CmdType.ForceLimit));

    CmdType.ReadActualForce             : CMD_TYPE_TO_STRING := StrReplace('ReadActualForce ({0})','{0}'            , UINT_TO_STRING(CmdType.ReadActualForce));

    CmdType.BrakeTest                   : CMD_TYPE_TO_STRING := StrReplace('BrakeTest ({0})','{0}'                  , UINT_TO_STRING(CmdType.BrakeTest));

    CmdType.SoftSwitchTCP               : CMD_TYPE_TO_STRING := StrReplace('SoftSwitchTCP ({0})','{0}'              , UINT_TO_STRING(CmdType.SoftSwitchTCP));

    CmdType.CreateSpline                : CMD_TYPE_TO_STRING := StrReplace('CreateSpline ({0})','{0}'               , UINT_TO_STRING(CmdType.CreateSpline));

    CmdType.DeleteSpline                : CMD_TYPE_TO_STRING := StrReplace('DeleteSpline ({0})','{0}'               , UINT_TO_STRING(CmdType.DeleteSpline));

    CmdType.MoveSpline                  : CMD_TYPE_TO_STRING := StrReplace('MoveSpline ({0})','{0}'                 , UINT_TO_STRING(CmdType.MoveSpline));

    CmdType.DynamicSpline               : CMD_TYPE_TO_STRING := StrReplace('DynamicSpline ({0})','{0}'              , UINT_TO_STRING(CmdType.DynamicSpline));

    CmdType.LoadMeasurementAutomatic    : CMD_TYPE_TO_STRING := StrReplace('LoadMeasurementAutomatic ({0})','{0}'   , UINT_TO_STRING(CmdType.LoadMeasurementAutomatic));

    CmdType.LoadMeasurementSequential   : CMD_TYPE_TO_STRING := StrReplace('LoadMeasurementSequential ({0})','{0}'  , UINT_TO_STRING(CmdType.LoadMeasurementSequential));

    CmdType.CollisionDetection          : CMD_TYPE_TO_STRING := StrReplace('CollisionDetection ({0})','{0}'         , UINT_TO_STRING(CmdType.CollisionDetection));

    CmdType.FreeDrive                   : CMD_TYPE_TO_STRING := StrReplace('FreeDrive ({0})','{0}'                  , UINT_TO_STRING(CmdType.FreeDrive));

    CmdType.UnitMeasurement             : CMD_TYPE_TO_STRING := StrReplace('UnitMeasurement ({0})','{0}'            , UINT_TO_STRING(CmdType.UnitMeasurement));

  ELSE
    CMD_TYPE_TO_STRING := CONCAT('CMD_TYPE_TO_STRING Function: Error -> no parsing for value',UINT_TO_STRING(Value));
  END_CASE

END_FUNCTION

(* ---- COLLISION_REACTION_MODE_TO_STRING.st ---- *)
FUNCTION COLLISION_REACTION_MODE_TO_STRING : STRING
// -------------------------------------------------------------------------
//  SRCI Robot Library
// -------------------------------------------------------------------------
//
//  Object:      COLLISION_REACTION_MODE_TO_STRING
//  Author:      Thorsten Brach
//  Date:        2025-01-24
//
//  Description:
//
//
//  Copyright:
//    (C) 2025 Thorsten Brach. All rights reserved
//             Licensed under the LGPL-3.0 license.
//
//  Disclaimer:
//    This project is provided without any guarantee and can be used for
//    private and commercial purposes. Any use is at the user’s
//    own risk and responsibility.
//
// -------------------------------------------------------------------------
VAR_INPUT
  /// CollisionReactionMode
  Value : CollisionReactionMode;
END_VAR

  CASE Value
  OF
    CollisionReactionMode.REVERSED_MOVEMENT : COLLISION_REACTION_MODE_TO_STRING := StrReplace('REVERSED_MOVEMENT ({0})','{0}' , USINT_TO_STRING(Value));
    CollisionReactionMode.STANDING_STILL    : COLLISION_REACTION_MODE_TO_STRING := StrReplace('STANDING_STILL ({0})'   ,'{0}' , USINT_TO_STRING(Value));
  ELSE
    COLLISION_REACTION_MODE_TO_STRING := CONCAT('COLLISION_REACTION_MODE_TO_STRING Function: Error -> no parsing for value ', USINT_TO_STRING(Value));
  END_CASE

END_FUNCTION

(* ---- CONNECTION_MODE_TO_STRING.st ---- *)
FUNCTION CONNECTION_MODE_TO_STRING : STRING
// -------------------------------------------------------------------------
//  SRCI Robot Library
// -------------------------------------------------------------------------
//
//  Object:      CONNECTION_MODE_TO_STRING
//  Author:      Thorsten Brach
//  Date:        2025-02-01
//
//  Description:
//
//
//  Copyright:
//    (C) 2025 Thorsten Brach. All rights reserved
//             Licensed under the LGPL-3.0 license.
//
//  Disclaimer:
//    This project is provided without any guarantee and can be used for
//    private and commercial purposes. Any use is at the user’s
//    own risk and responsibility.
//
// -------------------------------------------------------------------------
VAR_INPUT
  /// ConnectionMode
  Value : ConnectionMode;
END_VAR

  CASE Value
  OF
    ConnectionMode.RC_CONNECTED  : CONNECTION_MODE_TO_STRING := StrReplace('RC_CONNECTED ({0})'  ,'{0}' , SINT_TO_STRING(Value));
    ConnectionMode.PLC_CONNECTED : CONNECTION_MODE_TO_STRING := StrReplace('PLC_CONNECTED ({0})' ,'{0}' , SINT_TO_STRING(Value));
  ELSE
    CONNECTION_MODE_TO_STRING := CONCAT('CONNECTION_MODE_TO_STRING Function: Error -> no parsing for value ', SINT_TO_STRING(Value));
  END_CASE

END_FUNCTION

(* ---- CONVEYOR_TYPE_TO_STRING.st ---- *)
FUNCTION CONVEYOR_TYPE_TO_STRING : STRING
// -------------------------------------------------------------------------
//  SRCI Robot Library
// -------------------------------------------------------------------------
//
//  Object:      CONVEYOR_TYPE_TO_STRING
//  Author:      Thorsten Brach
//  Date:        2025-02-01
//
//  Description:
//
//
//  Copyright:
//    (C) 2025 Thorsten Brach. All rights reserved
//             Licensed under the LGPL-3.0 license.
//
//  Disclaimer:
//    This project is provided without any guarantee and can be used for
//    private and commercial purposes. Any use is at the user’s
//    own risk and responsibility.
//
// -------------------------------------------------------------------------
VAR_INPUT
  /// ConveyorType
  Value : ConveyorType;
END_VAR

  CASE Value
  OF
    ConveyorType.LINEAR_CONVEYOR_TRACKING   : CONVEYOR_TYPE_TO_STRING := StrReplace('LINEAR_CONVEYOR_TRACKING ({0})'   ,'{0}' , USINT_TO_STRING(Value));
    ConveyorType.CIRCULAR_CONVEYOR_TRACKING : CONVEYOR_TYPE_TO_STRING := StrReplace('CIRCULAR_CONVEYOR_TRACKING ({0})' ,'{0}' , USINT_TO_STRING(Value));
  ELSE
    CONVEYOR_TYPE_TO_STRING := CONCAT('CONVEYOR_TYPE_TO_STRING Function: Error -> no parsing for value ', USINT_TO_STRING(Value));
  END_CASE

END_FUNCTION

(* ---- DATA_ENABLE_SYNC_TO_STRING.st ---- *)
FUNCTION DATA_ENABLE_SYNC_TO_STRING : STRING
// -------------------------------------------------------------------------
//  SRCI Robot Library
// -------------------------------------------------------------------------
//
//  Object:      DATA_ENABLE_SYNC_TO_STRING
//  Author:      Thorsten Brach
//  Date:        2025-01-24
//
//  Description:
//
//
//  Copyright:
//    (C) 2025 Thorsten Brach. All rights reserved
//             Licensed under the LGPL-3.0 license.
//
//  Disclaimer:
//    This project is provided without any guarantee and can be used for
//    private and commercial purposes. Any use is at the user’s
//    own risk and responsibility.
//
// -------------------------------------------------------------------------
VAR_INPUT
  /// DataEnableSync
  Value : DataEnableSync;
END_VAR

VAR
  /// temporary byte
 _tmpByte : BYTE;
END_VAR

  _tmpByte.0 := Value.EnableSyncTool;
  _tmpByte.1 := Value.EnableSyncFrame;
  _tmpByte.2 := Value.EnableSyncLoad;
  _tmpByte.3 := Value.EnableSyncWorkArea;
  _tmpByte.4 := Value.EnableSyncSWLimits;
  _tmpByte.5 := Value.EnableSyncDefaultDynamics;
  _tmpByte.6 := Value.EnableSyncReferenceDynamics;

  DATA_ENABLE_SYNC_TO_STRING := BYTE_TO_STRING_BIN(_tmpByte);

END_FUNCTION

(* ---- DATA_IN_SYNC_TO_STRING.st ---- *)
FUNCTION DATA_IN_SYNC_TO_STRING : STRING
// -------------------------------------------------------------------------
//  SRCI Robot Library
// -------------------------------------------------------------------------
//
//  Object:      DATA_IN_SYNC_TO_STRING
//  Author:      Thorsten Brach
//  Date:        2025-01-24
//
//  Description:
//
//
//  Copyright:
//    (C) 2025 Thorsten Brach. All rights reserved
//             Licensed under the LGPL-3.0 license.
//
//  Disclaimer:
//    This project is provided without any guarantee and can be used for
//    private and commercial purposes. Any use is at the user’s
//    own risk and responsibility.
//
// -------------------------------------------------------------------------
VAR_INPUT
  /// DataInSync
  Value : DataInSync;
END_VAR

VAR
  /// temporary byte
 _tmpByte : BYTE;
END_VAR

  _tmpByte.0 := Value.ToolsInSync;
  _tmpByte.1 := Value.FramesInSync;
  _tmpByte.2 := Value.LoadsInSync;
  _tmpByte.3 := Value.WorkAreasInSync;
  _tmpByte.4 := Value.SoftwareLimitsInSync;
  _tmpByte.5 := Value.DefaultDynamicsInSync;
  _tmpByte.6 := Value.ReferenceDynamicsInSync;
  _tmpByte.7 := FALSE;

  DATA_IN_SYNC_TO_STRING := BYTE_TO_STRING_BIN(_tmpByte);

END_FUNCTION

(* ---- DATA_TYPE_TO_STRING.st ---- *)
FUNCTION DATA_TYPE_TO_STRING : STRING
// -------------------------------------------------------------------------
//  SRCI Robot Library
// -------------------------------------------------------------------------
//
//  Object:      DATA_TYPE_TO_STRING
//  Author:      Thorsten Brach
//  Date:        2025-03-05
//
//  Description:
//
//
//  Copyright:
//    (C) 2025 Thorsten Brach. All rights reserved
//             Licensed under the LGPL-3.0 license.
//
//  Disclaimer:
//    This project is provided without any guarantee and can be used for
//    private and commercial purposes. Any use is at the user’s
//    own risk and responsibility.
//
// -------------------------------------------------------------------------
VAR_INPUT
  /// DataType
  Value : DataType;
END_VAR

  CASE Value
  OF
    DataType.TYPE_BOOL       : DATA_TYPE_TO_STRING := StrReplace('BOOL ({0})'                ,'{0}' , USINT_TO_STRING(Value));
    DataType.TYPE_BYTE       : DATA_TYPE_TO_STRING := StrReplace('BYTE ({0})'                ,'{0}' , USINT_TO_STRING(Value));
    DataType.TYPE_WORD       : DATA_TYPE_TO_STRING := StrReplace('WORD ({0})'                ,'{0}' , USINT_TO_STRING(Value));
    DataType.TYPE_DWORD      : DATA_TYPE_TO_STRING := StrReplace('DWORD ({0})'               ,'{0}' , USINT_TO_STRING(Value));
    DataType.TYPE_SINT       : DATA_TYPE_TO_STRING := StrReplace('SINT ({0})'                ,'{0}' , USINT_TO_STRING(Value));
    DataType.TYPE_USINT      : DATA_TYPE_TO_STRING := StrReplace('USINT ({0})'               ,'{0}' , USINT_TO_STRING(Value));
    DataType.TYPE_INT        : DATA_TYPE_TO_STRING := StrReplace('INT ({0})'                 ,'{0}' , USINT_TO_STRING(Value));
    DataType.TYPE_UINT       : DATA_TYPE_TO_STRING := StrReplace('UINT ({0})'                ,'{0}' , USINT_TO_STRING(Value));
    DataType.TYPE_DINT       : DATA_TYPE_TO_STRING := StrReplace('DINT ({0})'                ,'{0}' , USINT_TO_STRING(Value));
    DataType.TYPE_UDINT      : DATA_TYPE_TO_STRING := StrReplace('UDINT ({0})'               ,'{0}' , USINT_TO_STRING(Value));
    DataType.TYPE_REAL       : DATA_TYPE_TO_STRING := StrReplace('REAL ({0})'                ,'{0}' , USINT_TO_STRING(Value));
    DataType.TYPE_CHAR       : DATA_TYPE_TO_STRING := StrReplace('CHAR ({0})'                ,'{0}' , USINT_TO_STRING(Value));
    DataType.TYPE_CHAR_ARRAY : DATA_TYPE_TO_STRING := StrReplace('ARRAY[0..3] OF CHAR ({0})' ,'{0}' , USINT_TO_STRING(Value));
  ELSE
    DATA_TYPE_TO_STRING := CONCAT('DATA_TYPE_TO_STRING Function: Error -> no parsing for value ', USINT_TO_STRING(Value));
  END_CASE

END_FUNCTION

(* ---- DEFINITION_MODE_TO_STRING.st ---- *)
FUNCTION DEFINITION_MODE_TO_STRING : STRING
// -------------------------------------------------------------------------
//  SRCI Robot Library
// -------------------------------------------------------------------------
//
//  Object:      DEFINITION_MODE_TO_STRING
//  Author:      Thorsten Brach
//  Date:        2025-02-01
//
//  Description:
//
//
//  Copyright:
//    (C) 2025 Thorsten Brach. All rights reserved
//             Licensed under the LGPL-3.0 license.
//
//  Disclaimer:
//    This project is provided without any guarantee and can be used for
//    private and commercial purposes. Any use is at the user’s
//    own risk and responsibility.
//
// -------------------------------------------------------------------------
VAR_INPUT
  /// DefinitionMode
  Value : DefinitionMode;
END_VAR

  CASE Value
  OF
    DefinitionMode.CENTER : DEFINITION_MODE_TO_STRING := StrReplace('CENTER ({0})','{0}' , USINT_TO_STRING(Value));
    DefinitionMode.FACE   : DEFINITION_MODE_TO_STRING := StrReplace('FACE ({0})'  ,'{0}' , USINT_TO_STRING(Value));
  ELSE
    DEFINITION_MODE_TO_STRING := CONCAT('DEFINITION_MODE_TO_STRING Function: Error -> no parsing for value ', USINT_TO_STRING(Value));
  END_CASE

END_FUNCTION

(* ---- DETECTION_MODE_TO_STRING.st ---- *)
FUNCTION DETECTION_MODE_TO_STRING : STRING
// -------------------------------------------------------------------------
//  SRCI Robot Library
// -------------------------------------------------------------------------
//
//  Object:      DETECTION_MODE_TO_STRING
//  Author:      Thorsten Brach
//  Date:        2025-02-01
//
//  Description:
//
//
//  Copyright:
//    (C) 2025 Thorsten Brach. All rights reserved
//             Licensed under the LGPL-3.0 license.
//
//  Disclaimer:
//    This project is provided without any guarantee and can be used for
//    private and commercial purposes. Any use is at the user’s
//    own risk and responsibility.
//
// -------------------------------------------------------------------------
VAR_INPUT
  /// DetectionMode
  Value : DetectionMode;
END_VAR

  CASE Value
  OF
    DetectionMode.TORQUE             : DETECTION_MODE_TO_STRING := StrReplace('TORQUE ({0})'             ,'{0}' , USINT_TO_STRING(Value));
    DetectionMode.FORCE              : DETECTION_MODE_TO_STRING := StrReplace('FORCE ({0})'              ,'{0}' , USINT_TO_STRING(Value));
    DetectionMode.ELECTRICAL_CURRENT : DETECTION_MODE_TO_STRING := StrReplace('ELECTRICAL_CURRENT ({0})' ,'{0}' , USINT_TO_STRING(Value));
    DetectionMode.FOLLOWING_ERROR    : DETECTION_MODE_TO_STRING := StrReplace('FOLLOWING_ERROR ({0})'    ,'{0}' , USINT_TO_STRING(Value));
  ELSE
    DETECTION_MODE_TO_STRING := CONCAT('DETECTION_MODE_TO_STRING Function: Error -> no parsing for value ', USINT_TO_STRING(Value));
  END_CASE

END_FUNCTION

(* ---- ERROR_REACTION_TO_STRING.st ---- *)
FUNCTION ERROR_REACTION_TO_STRING : STRING
// -------------------------------------------------------------------------
//  SRCI Robot Library
// -------------------------------------------------------------------------
//
//  Object:      ERROR_REACTION_TO_STRING
//  Author:      Thorsten Brach
//  Date:        2025-02-01
//
//  Description:
//
//
//  Copyright:
//    (C) 2025 Thorsten Brach. All rights reserved
//             Licensed under the LGPL-3.0 license.
//
//  Disclaimer:
//    This project is provided without any guarantee and can be used for
//    private and commercial purposes. Any use is at the user’s
//    own risk and responsibility.
//
// -------------------------------------------------------------------------
VAR_INPUT
  /// ErrorReaction
  Value : ErrorReaction;
END_VAR

  CASE Value
  OF
    ErrorReaction.ABORT_AND_MOVE : ERROR_REACTION_TO_STRING := StrReplace('ABORT_AND_MOVE ({0})','{0}' , USINT_TO_STRING(Value));
    ErrorReaction.ABORT          : ERROR_REACTION_TO_STRING := StrReplace('ABORT ({0})'         ,'{0}' , USINT_TO_STRING(Value));
    ErrorReaction.NO_REACTION    : ERROR_REACTION_TO_STRING := StrReplace('NO_REACTION ({0})'   ,'{0}' , USINT_TO_STRING(Value));
  ELSE
    ERROR_REACTION_TO_STRING := CONCAT('ERROR_REACTION_TO_STRING Function: Error -> no parsing for value ', USINT_TO_STRING(Value));
  END_CASE

END_FUNCTION

(* ---- ERROR_TRIGGER_MODE_TO_STRING.st ---- *)
FUNCTION ERROR_TRIGGER_MODE_TO_STRING : STRING
// -------------------------------------------------------------------------
//  SRCI Robot Library
// -------------------------------------------------------------------------
//
//  Object:      ERROR_TRIGGER_MODE_TO_STRING
//  Author:      Thorsten Brach
//  Date:        2025-02-01
//
//  Description:
//
//
//  Copyright:
//    (C) 2025 Thorsten Brach. All rights reserved
//             Licensed under the LGPL-3.0 license.
//
//  Disclaimer:
//    This project is provided without any guarantee and can be used for
//    private and commercial purposes. Any use is at the user’s
//    own risk and responsibility.
//
// -------------------------------------------------------------------------
VAR_INPUT
  /// ErrorTriggerMode
  Value : ErrorTriggerMode;
END_VAR

  CASE Value
  OF
    ErrorTriggerMode.ANY_COMMAND                    : ERROR_TRIGGER_MODE_TO_STRING := StrReplace('ANY_COMMAND ({0})'                    ,'{0}' , SINT_TO_STRING(Value));
    ErrorTriggerMode.GENERAL_COMMANDS               : ERROR_TRIGGER_MODE_TO_STRING := StrReplace('GENERAL_COMMANDS ({0})'               ,'{0}' , SINT_TO_STRING(Value));
    ErrorTriggerMode.ADMINISTRATIVE_COMMANDS        : ERROR_TRIGGER_MODE_TO_STRING := StrReplace('ADMINISTRATIVE_COMMANDS ({0})'        ,'{0}' , SINT_TO_STRING(Value));
    ErrorTriggerMode.MOVE_COMMANDS                  : ERROR_TRIGGER_MODE_TO_STRING := StrReplace('MOVE_COMMANDS ({0})'                  ,'{0}' , SINT_TO_STRING(Value));
    ErrorTriggerMode.PERIPHERY_COMMANDS             : ERROR_TRIGGER_MODE_TO_STRING := StrReplace('PERIPHERY_COMMANDS ({0})'             ,'{0}' , SINT_TO_STRING(Value));
    ErrorTriggerMode.EXTENDED_COMMANDS              : ERROR_TRIGGER_MODE_TO_STRING := StrReplace('EXTENDED_COMMANDS ({0})'              ,'{0}' , SINT_TO_STRING(Value));
    ErrorTriggerMode.SPECIFIC_COMMAND_OR_RI_MESSAGE : ERROR_TRIGGER_MODE_TO_STRING := StrReplace('SPECIFIC_COMMAND_OR_RI_MESSAGE ({0})' ,'{0}' , SINT_TO_STRING(Value));
    ErrorTriggerMode.SPECIFIC_RC_OR_RA_MESSAGE_CODE : ERROR_TRIGGER_MODE_TO_STRING := StrReplace('SPECIFIC_RC_OR_RA_MESSAGE_CODE ({0})' ,'{0}' , SINT_TO_STRING(Value));
    ErrorTriggerMode.ANY_RI_MESSAGE_CODE            : ERROR_TRIGGER_MODE_TO_STRING := StrReplace('ANY_RI_MESSAGE_CODE ({0})'            ,'{0}' , SINT_TO_STRING(Value));
    ErrorTriggerMode.ANY_RC_OR_RA_MESSAGE_CODE      : ERROR_TRIGGER_MODE_TO_STRING := StrReplace('ANY_RC_OR_RA_MESSAGE_CODE ({0})'      ,'{0}' , SINT_TO_STRING(Value));
  ELSE
    ERROR_TRIGGER_MODE_TO_STRING := CONCAT('ERROR_TRIGGER_MODE_TO_STRING Function: Error -> no parsing for value ', SINT_TO_STRING(Value));
  END_CASE

END_FUNCTION

(* ---- EXECUTION_MODE_TO_STRING.st ---- *)
FUNCTION EXECUTION_MODE_TO_STRING : STRING
// -------------------------------------------------------------------------
//  SRCI Robot Library
// -------------------------------------------------------------------------
//
//  Object:      EXECUTION_MODE_TO_STRING
//  Author:      Thorsten Brach
//  Date:        2025-01-20
//
//  Description:
//
//
//  Copyright:
//    (C) 2024 Thorsten Brach. All rights reserved
//             Licensed under the LGPL-3.0 license.
//
//  Disclaimer:
//    This project is provided without any guarantee and can be used for
//    private and commercial purposes. Any use is at the user’s
//    own risk and responsibility.
//
// -------------------------------------------------------------------------
VAR_INPUT
  /// ExecMode
  Value : ExecutionMode;
END_VAR

  CASE Value
  OF
    ExecutionMode.SEQUENCE_PRIMARY                 : EXECUTION_MODE_TO_STRING := StrReplace('SEQUENCE_PRIMARY ({0})'                 ,'{0}', USINT_TO_STRING(Value));
    ExecutionMode.SEQUENCE_ABORT_OTHERS_PRIMARY    : EXECUTION_MODE_TO_STRING := StrReplace('SEQUENCE_ABORT_OTHERS_PRIMARY ({0})'    ,'{0}', USINT_TO_STRING(Value));
    ExecutionMode.PARALLEL                         : EXECUTION_MODE_TO_STRING := StrReplace('PARALLEL ({0})'                         ,'{0}', USINT_TO_STRING(Value));
    ExecutionMode.CONTINUOUS                       : EXECUTION_MODE_TO_STRING := StrReplace('CONTINUOUS ({0})'                       ,'{0}', USINT_TO_STRING(Value));
    ExecutionMode.TRIGGER_MULTIPLE                 : EXECUTION_MODE_TO_STRING := StrReplace('TRIGGER_MULTIPLE ({0})'                 ,'{0}', USINT_TO_STRING(Value));
    ExecutionMode.SEQUENCE_SECONDARY               : EXECUTION_MODE_TO_STRING := StrReplace('SEQUENCE_SECONDARY ({0})'               ,'{0}', USINT_TO_STRING(Value));
    ExecutionMode.SEQUENCE_ABORT_OTHERS_SECONDARY  : EXECUTION_MODE_TO_STRING := StrReplace('SEQUENCE_ABORT_OTHERS_SECONDARY ({0})'  ,'{0}', USINT_TO_STRING(Value));
    ExecutionMode.STOP_PARALLEL_CONTINUOUS_TRIGGER : EXECUTION_MODE_TO_STRING := StrReplace('STOP_PARALLEL_CONTINUOUS_TRIGGER ({0})' ,'{0}', USINT_TO_STRING(Value));
  ELSE
    EXECUTION_MODE_TO_STRING := CONCAT('EXECUTION_MODE_TO_STRING Function: Error -> no parsing for value ', USINT_TO_STRING(Value));
  END_CASE

END_FUNCTION

(* ---- EXTERNAL_AXES_FLAGS_TO_STRING.st ---- *)
FUNCTION EXTERNAL_AXES_FLAGS_TO_STRING : STRING
// -------------------------------------------------------------------------
//  SRCI Robot Library
// -------------------------------------------------------------------------
//
//  Object:      EXTERNAL_AXES_FLAGS_TO_STRING
//  Author:      Thorsten Brach
//  Date:        2025-02-26
//
//  Description:
//
//
//  Copyright:
//    (C) 2025 Thorsten Brach. All rights reserved
//             Licensed under the LGPL-3.0 license.
//
//  Disclaimer:
//    This project is provided without any guarantee and can be used for
//    private and commercial purposes. Any use is at the user’s
//    own risk and responsibility.
//
// -------------------------------------------------------------------------
VAR_INPUT
  /// ExternalAxesFlags
  Value : ExternalAxesFlags;
END_VAR

VAR
 _tmpByte : BYTE;
END_VAR

  _tmpByte.0 := Value.Bit00;
  _tmpByte.1 := Value.AxisE1;
  _tmpByte.2 := Value.AxisE2;
  _tmpByte.3 := Value.AxisE3;
  _tmpByte.4 := Value.AxisE4;
  _tmpByte.5 := Value.AxisE5;
  _tmpByte.6 := Value.AxisE6;
  _tmpByte.7 := Value.Bit07;

  EXTERNAL_AXES_FLAGS_TO_STRING := BYTE_TO_STRING_BIN(_tmpByte);

END_FUNCTION

(* ---- FRAGMENT_ACTION_TO_STRING.st ---- *)
FUNCTION FRAGMENT_ACTION_TO_STRING : STRING
// -------------------------------------------------------------------------
//  SRCI Robot Library
// -------------------------------------------------------------------------
//
//  Object:      FRAGMENT_ACTION_TO_STRING
//  Author:      Thorsten Brach
//  Date:        2024-11-16
//
//  Description:
//
//
//  Copyright:
//    (C) 2024 Thorsten Brach. All rights reserved
//             Licensed under the LGPL-3.0 license.
//
//  Disclaimer:
//    This project is provided without any guarantee and can be used for
//    private and commercial purposes. Any use is at the user’s
//    own risk and responsibility.
//
// -------------------------------------------------------------------------
VAR_INPUT
  /// Fragment action
  FragmentAction : BYTE;
END_VAR

  IF ( FragmentAction.0 )
  THEN
   FRAGMENT_ACTION_TO_STRING := CONCAT(FRAGMENT_ACTION_TO_STRING, ' Complete (Bit 0)');
  END_IF

  IF ( FragmentAction.1 )
  THEN
   FRAGMENT_ACTION_TO_STRING := CONCAT(FRAGMENT_ACTION_TO_STRING, ' Reset (Bit 1)');
  END_IF

  IF ( FragmentAction.2 )
  THEN
   FRAGMENT_ACTION_TO_STRING := CONCAT(FRAGMENT_ACTION_TO_STRING, ' Clear (Bit 2)');
  END_IF

END_FUNCTION

(* ---- FRAME_CALCULATION_MODE_TO_STRING.st ---- *)
FUNCTION FRAME_CALCULATION_MODE_TO_STRING : STRING
// -------------------------------------------------------------------------
//  SRCI Robot Library
// -------------------------------------------------------------------------
//
//  Object:      FRAME_CALCULATION_MODE_TO_STRING
//  Author:      Thorsten Brach
//  Date:        2025-02-01
//
//  Description:
//
//
//  Copyright:
//    (C) 2025 Thorsten Brach. All rights reserved
//             Licensed under the LGPL-3.0 license.
//
//  Disclaimer:
//    This project is provided without any guarantee and can be used for
//    private and commercial purposes. Any use is at the user’s
//    own risk and responsibility.
//
// -------------------------------------------------------------------------
VAR_INPUT
  /// FrameCalculationMode
  Value : FrameCalculationMode;
END_VAR

  CASE Value
  OF
    FrameCalculationMode.THREE_POINT_METHOD : FRAME_CALCULATION_MODE_TO_STRING := StrReplace('THREE_POINT_METHOD ({0})','{0}' , SINT_TO_STRING(Value));
    FrameCalculationMode.FOUR_POINT_METHOD  : FRAME_CALCULATION_MODE_TO_STRING := StrReplace('FOUR_POINT_METHOD ({0})' ,'{0}' , SINT_TO_STRING(Value));
    FrameCalculationMode.ONE_POINT_METHOD   : FRAME_CALCULATION_MODE_TO_STRING := StrReplace('ONE_POINT_METHOD ({0})'  ,'{0}' , SINT_TO_STRING(Value));
  ELSE
    FRAME_CALCULATION_MODE_TO_STRING := CONCAT('FRAME_CALCULATION_MODE_TO_STRING Function: Error -> no parsing for value ', SINT_TO_STRING(Value));
  END_CASE

END_FUNCTION

(* ---- IEC_DATE_TO_STRING.st ---- *)
FUNCTION IEC_DATE_TO_STRING : STRING
// -------------------------------------------------------------------------
//  SRCI Robot Library
// -------------------------------------------------------------------------
//
//  Object:      IEC_DATE_TO_STRING
//  Author:      Thorsten Brach
//  Date:        2025-02-01
//
//  Description:
//
//
//  Copyright:
//    (C) 2025 Thorsten Brach. All rights reserved
//             Licensed under the LGPL-3.0 license.
//
//  Disclaimer:
//    This project is provided without any guarantee and can be used for
//    private and commercial purposes. Any use is at the user’s
//    own risk and responsibility.
//
// -------------------------------------------------------------------------
VAR_INPUT
  /// IEC Date
  Value : IEC_DATE;
END_VAR

VAR
  /// temporary date
 _tmpData : DATE;
END_VAR

  IEC_DATE_TO_STRING := DATE_TO_STRING(IEC_DATE_TO_DATE(Value));

END_FUNCTION

(* ---- IEC_TIME_TO_STRING.st ---- *)
FUNCTION IEC_TIME_TO_STRING : STRING
// -------------------------------------------------------------------------
//  SRCI Robot Library
// -------------------------------------------------------------------------
//
//  Object:      ORI_MODE_TO_STRING
//  Author:      Thorsten Brach
//  Date:        2025-01-24
//
//  Description:
//
//
//  Copyright:
//    (C) 2025 Thorsten Brach. All rights reserved
//             Licensed under the LGPL-3.0 license.
//
//  Disclaimer:
//    This project is provided without any guarantee and can be used for
//    private and commercial purposes. Any use is at the user’s
//    own risk and responsibility.
//
// -------------------------------------------------------------------------
VAR_INPUT
  /// IEC_TIME
  Value : IEC_TIME;
END_VAR
VAR
  /// temporary date
 _tmpData : DATE;
END_VAR

  IEC_TIME_TO_STRING := TOD_TO_STRING(IEC_TIME_TO_TIME(Value));

END_FUNCTION

(* ---- INTERPOLATION_MODE_TO_STRING.st ---- *)
FUNCTION INTERPOLATION_MODE_TO_STRING : STRING
// -------------------------------------------------------------------------
//  SRCI Robot Library
// -------------------------------------------------------------------------
//
//  Object:      INTERPOLATION_MODE_TO_STRING
//  Author:      Thorsten Brach
//  Date:        2025-02-01
//
//  Description:
//
//
//  Copyright:
//    (C) 2025 Thorsten Brach. All rights reserved
//             Licensed under the LGPL-3.0 license.
//
//  Disclaimer:
//    This project is provided without any guarantee and can be used for
//    private and commercial purposes. Any use is at the user’s
//    own risk and responsibility.
//
// -------------------------------------------------------------------------
VAR_INPUT
  /// InterpolationMode
  Value : InterpolationMode;
END_VAR

  CASE Value
  OF
    InterpolationMode.LINEAR_INTERPOLATION : INTERPOLATION_MODE_TO_STRING := StrReplace('LINEAR_INTERPOLATION ({0})' ,'{0}' , USINT_TO_STRING(Value));
    InterpolationMode.DIRECT_INTERPOLATION : INTERPOLATION_MODE_TO_STRING := StrReplace('DIRECT_INTERPOLATION ({0})' ,'{0}' , USINT_TO_STRING(Value));
  ELSE
    INTERPOLATION_MODE_TO_STRING := CONCAT('INTERPOLATION_MODE_TO_STRING Function: Error -> no parsing for value ', USINT_TO_STRING(Value));
  END_CASE

END_FUNCTION

(* ---- JOG_CONTROL_TO_STRING.st ---- *)
FUNCTION JOG_CONTROL_TO_STRING : STRING
// -------------------------------------------------------------------------
//  SRCI Robot Library
// -------------------------------------------------------------------------
//
//  Object:      JOG_CONTROL_TO_STRING
//  Author:      Thorsten Brach
//  Date:        2025-03-01
//
//  Description:
//
//
//  Copyright:
//    (C) 2025 Thorsten Brach. All rights reserved
//             Licensed under the LGPL-3.0 license.
//
//  Disclaimer:
//    This project is provided without any guarantee and can be used for
//    private and commercial purposes. Any use is at the user’s
//    own risk and responsibility.
//
// -------------------------------------------------------------------------
VAR_INPUT
  /// JogControl
  Value : JogControl;
END_VAR

  JOG_CONTROL_TO_STRING := '2#';

  IF (Value.E6_Neg)
  THEN
    JOG_CONTROL_TO_STRING := CONCAT(JOG_CONTROL_TO_STRING, '1');
  ELSE
    JOG_CONTROL_TO_STRING := CONCAT(JOG_CONTROL_TO_STRING, '0');
  END_IF

  IF (Value.E6_Pos)
  THEN
    JOG_CONTROL_TO_STRING := CONCAT(JOG_CONTROL_TO_STRING, '1');
  ELSE
    JOG_CONTROL_TO_STRING := CONCAT(JOG_CONTROL_TO_STRING, '0');
  END_IF

  IF (Value.E5_Neg)
  THEN
    JOG_CONTROL_TO_STRING := CONCAT(JOG_CONTROL_TO_STRING, '1');
  ELSE
    JOG_CONTROL_TO_STRING := CONCAT(JOG_CONTROL_TO_STRING, '0');
  END_IF

  IF (Value.E5_Pos)
  THEN
    JOG_CONTROL_TO_STRING := CONCAT(JOG_CONTROL_TO_STRING, '1_');
  ELSE
    JOG_CONTROL_TO_STRING := CONCAT(JOG_CONTROL_TO_STRING, '0_');
  END_IF

  IF (Value.E4_Neg)
  THEN
    JOG_CONTROL_TO_STRING := CONCAT(JOG_CONTROL_TO_STRING, '1');
  ELSE
    JOG_CONTROL_TO_STRING := CONCAT(JOG_CONTROL_TO_STRING, '0');
  END_IF

  IF (Value.E4_Pos)
  THEN
    JOG_CONTROL_TO_STRING := CONCAT(JOG_CONTROL_TO_STRING, '1');
  ELSE
    JOG_CONTROL_TO_STRING := CONCAT(JOG_CONTROL_TO_STRING, '0');
  END_IF

  IF (Value.E3_Neg)
  THEN
    JOG_CONTROL_TO_STRING := CONCAT(JOG_CONTROL_TO_STRING, '1');
  ELSE
    JOG_CONTROL_TO_STRING := CONCAT(JOG_CONTROL_TO_STRING, '0');
  END_IF

  IF (Value.E3_Pos)
  THEN
    JOG_CONTROL_TO_STRING := CONCAT(JOG_CONTROL_TO_STRING, '1');
  ELSE
    JOG_CONTROL_TO_STRING := CONCAT(JOG_CONTROL_TO_STRING, '0');
  END_IF

  JOG_CONTROL_TO_STRING := CONCAT(JOG_CONTROL_TO_STRING, '_');

  IF (Value.E2_Neg)
  THEN
    JOG_CONTROL_TO_STRING := CONCAT(JOG_CONTROL_TO_STRING, '1');
  ELSE
    JOG_CONTROL_TO_STRING := CONCAT(JOG_CONTROL_TO_STRING, '0');
  END_IF

  IF (Value.E2_Pos)
  THEN
    JOG_CONTROL_TO_STRING := CONCAT(JOG_CONTROL_TO_STRING, '1');
  ELSE
    JOG_CONTROL_TO_STRING := CONCAT(JOG_CONTROL_TO_STRING, '0');
  END_IF

  IF (Value.E1_Neg)
  THEN
    JOG_CONTROL_TO_STRING := CONCAT(JOG_CONTROL_TO_STRING, '1');
  ELSE
    JOG_CONTROL_TO_STRING := CONCAT(JOG_CONTROL_TO_STRING, '0');
  END_IF

  IF (Value.E1_Pos)
  THEN
    JOG_CONTROL_TO_STRING := CONCAT(JOG_CONTROL_TO_STRING, '1');
  ELSE
    JOG_CONTROL_TO_STRING := CONCAT(JOG_CONTROL_TO_STRING, '0');
  END_IF

  IF (Value.Rz_J6_Neg)
  THEN
    JOG_CONTROL_TO_STRING := CONCAT(JOG_CONTROL_TO_STRING, '1');
  ELSE
    JOG_CONTROL_TO_STRING := CONCAT(JOG_CONTROL_TO_STRING, '0');
  END_IF

  IF (Value.Rz_J6_Pos)
  THEN
    JOG_CONTROL_TO_STRING := CONCAT(JOG_CONTROL_TO_STRING, '1');
  ELSE
    JOG_CONTROL_TO_STRING := CONCAT(JOG_CONTROL_TO_STRING, '0');
  END_IF

  IF (Value.Ry_J5_Neg)
  THEN
    JOG_CONTROL_TO_STRING := CONCAT(JOG_CONTROL_TO_STRING, '1');
  ELSE
    JOG_CONTROL_TO_STRING := CONCAT(JOG_CONTROL_TO_STRING, '0');
  END_IF

  IF (Value.Ry_J5_Pos)
  THEN
    JOG_CONTROL_TO_STRING := CONCAT(JOG_CONTROL_TO_STRING, '1');
  ELSE
    JOG_CONTROL_TO_STRING := CONCAT(JOG_CONTROL_TO_STRING, '0');
  END_IF

  JOG_CONTROL_TO_STRING := CONCAT(JOG_CONTROL_TO_STRING, '_');

  IF (Value.Rx_J4_Neg)
  THEN
    JOG_CONTROL_TO_STRING := CONCAT(JOG_CONTROL_TO_STRING, '1');
  ELSE
    JOG_CONTROL_TO_STRING := CONCAT(JOG_CONTROL_TO_STRING, '0');
  END_IF

  IF (Value.Rx_J4_Pos)
  THEN
    JOG_CONTROL_TO_STRING := CONCAT(JOG_CONTROL_TO_STRING, '1');
  ELSE
    JOG_CONTROL_TO_STRING := CONCAT(JOG_CONTROL_TO_STRING, '0');
  END_IF

  IF (Value.Z_J3_Neg)
  THEN
    JOG_CONTROL_TO_STRING := CONCAT(JOG_CONTROL_TO_STRING, '1');
  ELSE
    JOG_CONTROL_TO_STRING := CONCAT(JOG_CONTROL_TO_STRING, '0');
  END_IF

  IF (Value.Z_J3_Pos)
  THEN
    JOG_CONTROL_TO_STRING := CONCAT(JOG_CONTROL_TO_STRING, '1');
  ELSE
    JOG_CONTROL_TO_STRING := CONCAT(JOG_CONTROL_TO_STRING, '0');
  END_IF

  IF (Value.Y_J2_Neg)
  THEN
    JOG_CONTROL_TO_STRING := CONCAT(JOG_CONTROL_TO_STRING, '1');
  ELSE
    JOG_CONTROL_TO_STRING := CONCAT(JOG_CONTROL_TO_STRING, '0');
  END_IF

  IF (Value.Y_J2_Pos)
  THEN
    JOG_CONTROL_TO_STRING := CONCAT(JOG_CONTROL_TO_STRING, '1');
  ELSE
    JOG_CONTROL_TO_STRING := CONCAT(JOG_CONTROL_TO_STRING, '0');
  END_IF

  IF (Value.X_J1_Neg)
  THEN
    JOG_CONTROL_TO_STRING := CONCAT(JOG_CONTROL_TO_STRING, '1');
  ELSE
    JOG_CONTROL_TO_STRING := CONCAT(JOG_CONTROL_TO_STRING, '0');
  END_IF

  IF (Value.X_J1_Pos)
  THEN
    JOG_CONTROL_TO_STRING := CONCAT(JOG_CONTROL_TO_STRING, '1');
  ELSE
    JOG_CONTROL_TO_STRING := CONCAT(JOG_CONTROL_TO_STRING, '0');
  END_IF

END_FUNCTION

(* ---- JOG_MODE_TO_STRING.st ---- *)
FUNCTION JOG_MODE_TO_STRING : STRING
// -------------------------------------------------------------------------
//  SRCI Robot Library
// -------------------------------------------------------------------------
//
//  Object:      JOG_MODE_TO_STRING
//  Author:      Thorsten Brach
//  Date:        2025-01-20
//
//  Description:
//
//
//  Copyright:
//    (C) 2025 Thorsten Brach. All rights reserved
//             Licensed under the LGPL-3.0 license.
//
//  Disclaimer:
//    This project is provided without any guarantee and can be used for
//    private and commercial purposes. Any use is at the user’s
//    own risk and responsibility.
//
// -------------------------------------------------------------------------
VAR_INPUT
  /// JogMode
  Value : JogMode;
END_VAR

  CASE Value
  OF
    JogMode.JOG_FRAME : JOG_MODE_TO_STRING := StrReplace('JOG_FRAME ({0})','{0}' , USINT_TO_STRING(Value));
    JogMode.JOG_TOOL  : JOG_MODE_TO_STRING := StrReplace('JOG_TOOL ({0})','{0}'  , USINT_TO_STRING(Value));
    JogMode.JOG_AXES  : JOG_MODE_TO_STRING := StrReplace('JOG_AXES ({0})','{0}'  , USINT_TO_STRING(Value));
  ELSE
    JOG_MODE_TO_STRING := CONCAT('JOG_MODE_TO_STRING Function: Error -> no parsing for value ', USINT_TO_STRING(Value));
  END_CASE

END_FUNCTION

(* ---- LIMIT_MODE_TO_STRING.st ---- *)
FUNCTION LIMIT_MODE_TO_STRING : STRING
// -------------------------------------------------------------------------
//  SRCI Robot Library
// -------------------------------------------------------------------------
//
//  Object:      LIMIT_MODE_TO_STRING
//  Author:      Thorsten Brach
//  Date:        2025-01-24
//
//  Description:
//
//
//  Copyright:
//    (C) 2025 Thorsten Brach. All rights reserved
//             Licensed under the LGPL-3.0 license.
//
//  Disclaimer:
//    This project is provided without any guarantee and can be used for
//    private and commercial purposes. Any use is at the user’s
//    own risk and responsibility.
//
// -------------------------------------------------------------------------
VAR_INPUT
  /// LimitMode
  Value : LimitMode;
END_VAR

  CASE Value
  OF
    LimitMode.LIMIT_DEFINED    : LIMIT_MODE_TO_STRING := StrReplace('LIMIT_DEFINED ({0})'    ,'{0}' , USINT_TO_STRING(Value));
    LimitMode.NO_LIMIT_DEFINED : LIMIT_MODE_TO_STRING := StrReplace('NO_LIMIT_DEFINED ({0})' ,'{0}' , USINT_TO_STRING(Value));
  ELSE
    LIMIT_MODE_TO_STRING := CONCAT('LIMIT_MODE_TO_STRING Function: Error -> no parsing for value ', USINT_TO_STRING(Value));
  END_CASE

END_FUNCTION

(* ---- LOAD_MEASUREMENT_MODE_TO_STRING.st ---- *)
FUNCTION LOAD_MEASUREMENT_MODE_TO_STRING : STRING
// -------------------------------------------------------------------------
//  SRCI Robot Library
// -------------------------------------------------------------------------
//
//  Object:      LOAD_MEASUREMENT_MODE_TO_STRING
//  Author:      Thorsten Brach
//  Date:        2025-02-01
//
//  Description:
//
//
//  Copyright:
//    (C) 2025 Thorsten Brach. All rights reserved
//             Licensed under the LGPL-3.0 license.
//
//  Disclaimer:
//    This project is provided without any guarantee and can be used for
//    private and commercial purposes. Any use is at the user’s
//    own risk and responsibility.
//
// -------------------------------------------------------------------------
VAR_INPUT
  /// LoadMeasurementMode
  Value : LoadMeasurementMode;
END_VAR

  CASE Value
  OF
    LoadMeasurementMode.ONE_POSITION         : LOAD_MEASUREMENT_MODE_TO_STRING := StrReplace('ONE_POSITION ({0})'        ,'{0}' , USINT_TO_STRING(Value));
    LoadMeasurementMode.CONFIGURATION_ANGLE  : LOAD_MEASUREMENT_MODE_TO_STRING := StrReplace('CONFIGURATION_ANGLE ({0})' ,'{0}' , USINT_TO_STRING(Value));
    LoadMeasurementMode.AREA                 : LOAD_MEASUREMENT_MODE_TO_STRING := StrReplace('AREA ({0})'                ,'{0}' , USINT_TO_STRING(Value));
    LoadMeasurementMode.TWO_POSITIONS        : LOAD_MEASUREMENT_MODE_TO_STRING := StrReplace('TWO_POSITIONS ({0})'       ,'{0}' , USINT_TO_STRING(Value));
  ELSE
    LOAD_MEASUREMENT_MODE_TO_STRING := CONCAT('LOAD_MEASUREMENT_MODE_TO_STRING Function: Error -> no parsing for value ', USINT_TO_STRING(Value));
  END_CASE

END_FUNCTION

(* ---- LOAD_MEASUREMENT_STEPS_TO_STRING.st ---- *)
FUNCTION LOAD_MEASUREMENT_STEPS_TO_STRING : STRING
// -------------------------------------------------------------------------
//  SRCI Robot Library
// -------------------------------------------------------------------------
//
//  Object:      LOAD_MEASUREMENT_STEPS_TO_STRING
//  Author:      Thorsten Brach
//  Date:        2025-02-01
//
//  Description:
//
//
//  Copyright:
//    (C) 2025 Thorsten Brach. All rights reserved
//             Licensed under the LGPL-3.0 license.
//
//  Disclaimer:
//    This project is provided without any guarantee and can be used for
//    private and commercial purposes. Any use is at the user’s
//    own risk and responsibility.
//
// -------------------------------------------------------------------------
VAR_INPUT
  /// LoadMeasurementSteps
  Value : LoadMeasurementSteps;
END_VAR

  CASE Value
  OF
    LoadMeasurementSteps.RESET            : LOAD_MEASUREMENT_STEPS_TO_STRING := StrReplace('RESET ({0})'            ,'{0}' , USINT_TO_STRING(Value));
    LoadMeasurementSteps.FIRST_POSITION   : LOAD_MEASUREMENT_STEPS_TO_STRING := StrReplace('FIRST_POSITION ({0})'   ,'{0}' , USINT_TO_STRING(Value));
    LoadMeasurementSteps.SECOND_POSITION  : LOAD_MEASUREMENT_STEPS_TO_STRING := StrReplace('SECOND_POSITION ({0})'  ,'{0}' , USINT_TO_STRING(Value));
    LoadMeasurementSteps.THIRD_POSITION   : LOAD_MEASUREMENT_STEPS_TO_STRING := StrReplace('THIRD_POSITION ({0})'   ,'{0}' , USINT_TO_STRING(Value));
    LoadMeasurementSteps.FOURTH_POSITION  : LOAD_MEASUREMENT_STEPS_TO_STRING := StrReplace('FOURTH_POSITION ({0})'  ,'{0}' , USINT_TO_STRING(Value));
    LoadMeasurementSteps.LOAD_CALCULATION : LOAD_MEASUREMENT_STEPS_TO_STRING := StrReplace('LOAD_CALCULATION ({0})' ,'{0}' , USINT_TO_STRING(Value));
  ELSE
    LOAD_MEASUREMENT_STEPS_TO_STRING := CONCAT('LOAD_MEASUREMENT_STEPS_TO_STRING Function: Error -> no parsing for value ', USINT_TO_STRING(Value));
  END_CASE

END_FUNCTION

(* ---- LOG_LEVEL_TO_STRING.st ---- *)
FUNCTION LOG_LEVEL_TO_STRING : STRING
// -------------------------------------------------------------------------
//  SRCI Robot Library
// -------------------------------------------------------------------------
//
//  Object:      LOG_LEVEL_TO_STRING
//  Author:      Thorsten Brach
//  Date:        2025-01-24
//
//  Description:
//
//
//  Copyright:
//    (C) 2025 Thorsten Brach. All rights reserved
//             Licensed under the LGPL-3.0 license.
//
//  Disclaimer:
//    This project is provided without any guarantee and can be used for
//    private and commercial purposes. Any use is at the user’s
//    own risk and responsibility.
//
// -------------------------------------------------------------------------
VAR_INPUT
  /// LogLevel
  Value : LogLevel;
END_VAR

  CASE Value
  OF
    LogLevel.DEACTIVATE  : LOG_LEVEL_TO_STRING := StrReplace('DEACTIVATE ({0})' ,'{0}' , SINT_TO_STRING(Value));
    LogLevel.DEBUG       : LOG_LEVEL_TO_STRING := StrReplace('DEBUG ({0})'      ,'{0}' , SINT_TO_STRING(Value));
    LogLevel.INFO        : LOG_LEVEL_TO_STRING := StrReplace('INFO ({0})'       ,'{0}' , SINT_TO_STRING(Value));
    LogLevel.WARNING     : LOG_LEVEL_TO_STRING := StrReplace('WARNING ({0})'    ,'{0}' , SINT_TO_STRING(Value));
    LogLevel.ERROR       : LOG_LEVEL_TO_STRING := StrReplace('ERROR ({0})'      ,'{0}' , SINT_TO_STRING(Value));
    LogLevel.FATAL_ERROR : LOG_LEVEL_TO_STRING := StrReplace('FATAL_ERROR ({0})','{0}' , SINT_TO_STRING(Value));
  ELSE
    LOG_LEVEL_TO_STRING := CONCAT('LOG_LEVEL_TO_STRING Function: Error -> no parsing for value ', SINT_TO_STRING(Value));
  END_CASE

END_FUNCTION

(* ---- LOGON_MODE_TO_STRING.st ---- *)
FUNCTION LOGON_MODE_TO_STRING : STRING
// -------------------------------------------------------------------------
//  SRCI Robot Library
// -------------------------------------------------------------------------
//
//  Object:      LOGON_MODE_TO_STRING
//  Author:      Thorsten Brach
//  Date:        2025-02-01
//
//  Description:
//
//
//  Copyright:
//    (C) 2025 Thorsten Brach. All rights reserved
//             Licensed under the LGPL-3.0 license.
//
//  Disclaimer:
//    This project is provided without any guarantee and can be used for
//    private and commercial purposes. Any use is at the user’s
//    own risk and responsibility.
//
// -------------------------------------------------------------------------
VAR_INPUT
  /// LogonMode
  Value : LogonMode;
END_VAR

  CASE Value
  OF
    LogonMode.PASSWORD_ONLY         : LOGON_MODE_TO_STRING := StrReplace('PASSWORD_ONLY ({0})'         ,'{0}' , SINT_TO_STRING(Value));
    LogonMode.USERNAME_AND_PASSWORD : LOGON_MODE_TO_STRING := StrReplace('USERNAME_AND_PASSWORD ({0})' ,'{0}' , SINT_TO_STRING(Value));
    LogonMode.LEVEL_ID_AND_PASSWORD : LOGON_MODE_TO_STRING := StrReplace('LEVEL_ID_AND_PASSWORD ({0})' ,'{0}' , SINT_TO_STRING(Value));
  ELSE
    LOGON_MODE_TO_STRING := CONCAT('LOGON_MODE_TO_STRING Function: Error -> no parsing for value ', SINT_TO_STRING(Value));
  END_CASE

END_FUNCTION

(* ---- MEASUREING_UNIT_MODE_TO_STRING.st ---- *)
FUNCTION MEASUREING_UNIT_MODE_TO_STRING : STRING
// -------------------------------------------------------------------------
//  SRCI Robot Library
// -------------------------------------------------------------------------
//
//  Object:      MEASUREING_UNIT_MODE_TO_STRING
//  Author:      Thorsten Brach
//  Date:        2025-01-24
//
//  Description:
//
//
//  Copyright:
//    (C) 2025 Thorsten Brach. All rights reserved
//             Licensed under the LGPL-3.0 license.
//
//  Disclaimer:
//    This project is provided without any guarantee and can be used for
//    private and commercial purposes. Any use is at the user’s
//    own risk and responsibility.
//
// -------------------------------------------------------------------------
VAR_INPUT
  /// MeasuringUnitMode
  Value : MeasuringUnitMode;
END_VAR

  CASE Value
  OF
    MeasuringUnitMode.VECTOR_LENGTH  : MEASUREING_UNIT_MODE_TO_STRING := StrReplace('VECTOR_LENGTH ({0})'  ,'{0}' , USINT_TO_STRING(Value));
    MeasuringUnitMode.SEGMENT_LENGTH : MEASUREING_UNIT_MODE_TO_STRING := StrReplace('SEGMENT_LENGTH ({0})' ,'{0}' , USINT_TO_STRING(Value));
    MeasuringUnitMode.TIME_DURATION  : MEASUREING_UNIT_MODE_TO_STRING := StrReplace('TIME_DURATION ({0})'  ,'{0}' , USINT_TO_STRING(Value));
  ELSE
    MEASUREING_UNIT_MODE_TO_STRING := CONCAT('MEASUREING_UNIT_MODE_TO_STRING Function: Error -> no parsing for value ', USINT_TO_STRING(Value));
  END_CASE

END_FUNCTION

(* ---- MEASURING_IO_MODE_TO_STRING.st ---- *)
FUNCTION MEASURING_IO_MODE_TO_STRING : STRING
// -------------------------------------------------------------------------
//  SRCI Robot Library
// -------------------------------------------------------------------------
//
//  Object:      MEASURING_IO_MODE_TO_STRING
//  Author:      Thorsten Brach
//  Date:        2025-02-23
//
//  Description:
//
//
//  Copyright:
//    (C) 2025 Thorsten Brach. All rights reserved
//             Licensed under the LGPL-3.0 license.
//
//  Disclaimer:
//    This project is provided without any guarantee and can be used for
//    private and commercial purposes. Any use is at the user’s
//    own risk and responsibility.
//
// -------------------------------------------------------------------------
VAR_INPUT
  /// MeasuringIoMode
  Value : MeasuringIoMode;
END_VAR

  CASE Value
  OF
    MeasuringIoMode.MEASUREMENT_AT_NEXT_RISING_EDGE             : MEASURING_IO_MODE_TO_STRING := StrReplace('MEASUREMENT_AT_NEXT_RISING_EDGE ({0})'             ,'{0}' , USINT_TO_STRING(Value));
    MeasuringIoMode.MEASUREMENT_AT_NEXT_FALLING_EDGE            : MEASURING_IO_MODE_TO_STRING := StrReplace('MEASUREMENT_AT_NEXT_FALLING_EDGE ({0})'            ,'{0}' , USINT_TO_STRING(Value));
    MeasuringIoMode.MEASUREMENT_AT_NEXT_EDGE                    : MEASURING_IO_MODE_TO_STRING := StrReplace('MEASUREMENT_AT_NEXT_EDGE ({0})'                    ,'{0}' , USINT_TO_STRING(Value));
    MeasuringIoMode.MEASUREMENT_AT_TWO_EDGES_BEGIN_WITH_RISING  : MEASURING_IO_MODE_TO_STRING := StrReplace('MEASUREMENT_AT_TWO_EDGES_BEGIN_WITH_RISING ({0})'  ,'{0}' , USINT_TO_STRING(Value));
    MeasuringIoMode.MEASUREMENT_AT_TWO_EDGES_BEGIN_WITH_FALLING : MEASURING_IO_MODE_TO_STRING := StrReplace('MEASUREMENT_AT_TWO_EDGES_BEGIN_WITH_FALLING ({0})' ,'{0}' , USINT_TO_STRING(Value));
  ELSE
    MEASURING_IO_MODE_TO_STRING := CONCAT('MEASURING_IO_MODE_TO_STRING Function: Error -> no parsing for value ', USINT_TO_STRING(Value));
  END_CASE

END_FUNCTION

(* ---- MEASURING_UNIT_MODE_TO_STRING.st ---- *)
FUNCTION MEASURING_UNIT_MODE_TO_STRING : STRING
// -------------------------------------------------------------------------
//  SRCI Robot Library
// -------------------------------------------------------------------------
//
//  Object:      MEASURING_UNIT_MODE_TO_STRING
//  Author:      Thorsten Brach
//  Date:        2025-02-26
//
//  Description:
//
//
//  Copyright:
//    (C) 2025 Thorsten Brach. All rights reserved
//             Licensed under the LGPL-3.0 license.
//
//  Disclaimer:
//    This project is provided without any guarantee and can be used for
//    private and commercial purposes. Any use is at the user’s
//    own risk and responsibility.
//
// -------------------------------------------------------------------------
VAR_INPUT
  /// MeasuringUnitMode
  Value : MeasuringUnitMode;
END_VAR

  CASE Value
  OF
    MeasuringUnitMode.VECTOR_LENGTH   : MEASURING_UNIT_MODE_TO_STRING := StrReplace('VECTOR_LENGTH ({0})'  ,'{0}' , USINT_TO_STRING(Value));
    MeasuringUnitMode.SEGMENT_LENGTH  : MEASURING_UNIT_MODE_TO_STRING := StrReplace('SEGMENT_LENGTH ({0})' ,'{0}' , USINT_TO_STRING(Value));
    MeasuringUnitMode.TIME_DURATION   : MEASURING_UNIT_MODE_TO_STRING := StrReplace('TIME_DURATION ({0})'  ,'{0}' , USINT_TO_STRING(Value));
  ELSE
    MEASURING_UNIT_MODE_TO_STRING := CONCAT('MEASURING_UNIT_MODE_TO_STRING Function: Error -> no parsing for value ', USINT_TO_STRING(Value));
  END_CASE

END_FUNCTION
